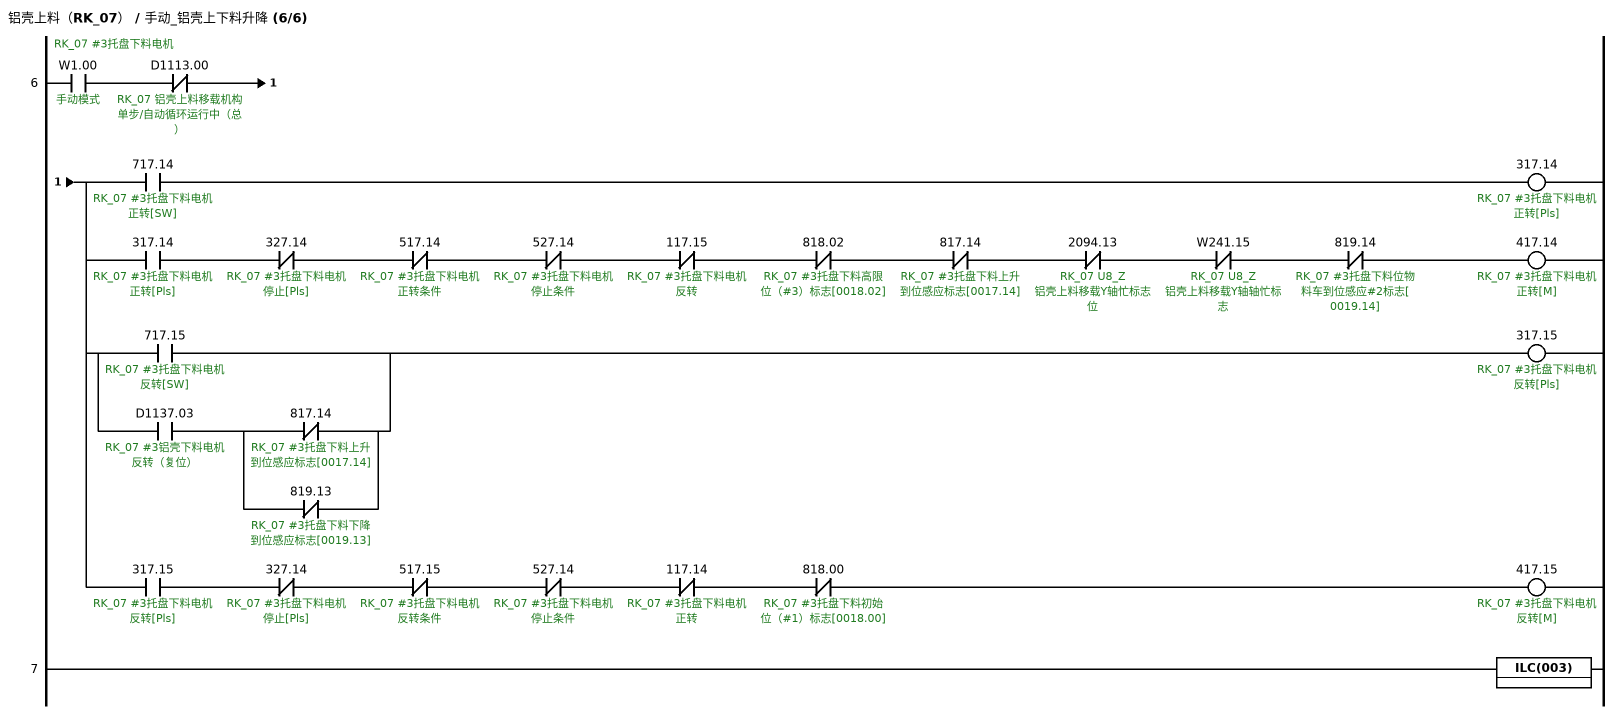
; [picture p576: 铝壳上料（RK_07） / 手动_铝壳上下料升降, rungs 6-7]
; rung 6: RK_07 #3托盘下料电机
LD W1.00  ; 手动模式
ANDNOT D1113.00  ; RK_07 铝壳上料移载机构单步/自动循环运行中（总）
OUT TR0
AND 717.14  ; RK_07 #3托盘下料电机正转[SW]
OUT 317.14  ; RK_07 #3托盘下料电机正转[Pls]
LD TR0
AND 317.14  ; RK_07 #3托盘下料电机正转[Pls]
ANDNOT 327.14  ; RK_07 #3托盘下料电机停止[Pls]
ANDNOT 517.14  ; RK_07 #3托盘下料电机正转条件
ANDNOT 527.14  ; RK_07 #3托盘下料电机停止条件
ANDNOT 117.15  ; RK_07 #3托盘下料电机反转
ANDNOT 818.02  ; RK_07 #3托盘下料高限位（#3）标志[0018.02]
ANDNOT 817.14  ; RK_07 #3托盘下料上升到位感应标志[0017.14]  // 手动模式加此联锁！
ANDNOT 2094.13  ; RK_07 U8_Z 铝壳上料移载Y轴忙标志位
ANDNOT W241.15  ; RK_07 U8_Z 铝壳上料移载Y轴轴忙标志
ANDNOT 819.14  ; RK_07 #3托盘下料位物料车到位感应#2标志[0019.14]
OUT 417.14  ; RK_07 #3托盘下料电机正转[M]
LD TR0
LD 717.15  ; RK_07 #3托盘下料电机反转[SW]
LD D1137.03  ; RK_07 #3铝壳下料电机反转（复位）
LDNOT 817.14  ; RK_07 #3托盘下料上升到位感应标志[0017.14]
ORNOT 819.13  ; RK_07 #3托盘下料下降到位感应标志[0019.13]
ANDLD
ORLD
ANDLD
OUT 317.15  ; RK_07 #3托盘下料电机反转[Pls]
LD TR0
AND 317.15  ; RK_07 #3托盘下料电机反转[Pls]
ANDNOT 327.14  ; RK_07 #3托盘下料电机停止[Pls]
ANDNOT 517.15  ; RK_07 #3托盘下料电机反转条件
ANDNOT 527.14  ; RK_07 #3托盘下料电机停止条件
ANDNOT 117.14  ; RK_07 #3托盘下料电机正转
ANDNOT 818.00  ; RK_07 #3托盘下料初始位（#1）标志[0018.00]
OUT 417.15  ; RK_07 #3托盘下料电机反转[M]
; rung 7
ILC(003)

### Section 自动_铝壳进料

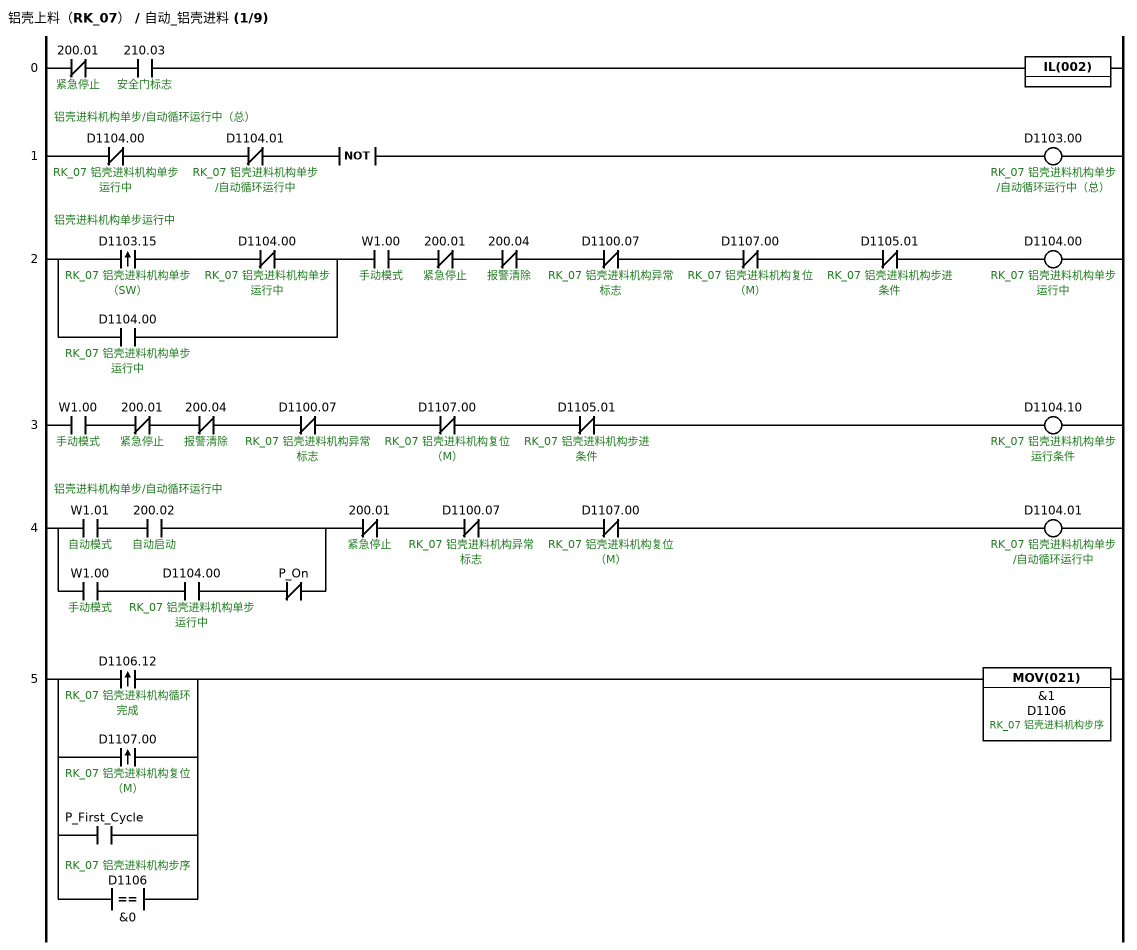
; rung 0
LDNOT 200.01  ; 紧急停止
AND 210.03  ; 安全门标志
IL(002)
; rung 1: 铝壳进料机构单步/自动循环运行中（总）
LDNOT D1104.00  ; RK_07 铝壳进料机构单步运行中
ANDNOT D1104.01  ; RK_07 铝壳进料机构单步/自动循环运行中
NOT(520)
OUT D1103.00  ; RK_07 铝壳进料机构单步/自动循环运行中（总）
; rung 2: 铝壳进料机构单步运行中
@LD D1103.15  ; RK_07 铝壳进料机构单步（SW）
ANDNOT D1104.00  ; RK_07 铝壳进料机构单步运行中
OR D1104.00  ; RK_07 铝壳进料机构单步运行中
AND W1.00  ; 手动模式
ANDNOT 200.01  ; 紧急停止
ANDNOT 200.04  ; 报警清除
ANDNOT D1100.07  ; RK_07 铝壳进料机构异常标志
ANDNOT D1107.00  ; RK_07 铝壳进料机构复位（M）
ANDNOT D1105.01  ; RK_07 铝壳进料机构步进条件
OUT D1104.00  ; RK_07 铝壳进料机构单步运行中
; rung 3
LD W1.00  ; 手动模式
ANDNOT 200.01  ; 紧急停止
ANDNOT 200.04  ; 报警清除
ANDNOT D1100.07  ; RK_07 铝壳进料机构异常标志
ANDNOT D1107.00  ; RK_07 铝壳进料机构复位（M）
ANDNOT D1105.01  ; RK_07 铝壳进料机构步进条件
OUT D1104.10  ; RK_07 铝壳进料机构单步运行条件
; rung 4: 铝壳进料机构单步/自动循环运行中
LD W1.01  ; 自动模式
AND 200.02  ; 自动启动
LD W1.00  ; 手动模式
AND D1104.00  ; RK_07 铝壳进料机构单步运行中
ANDNOT P_On
ORLD
ANDNOT 200.01  ; 紧急停止
ANDNOT D1100.07  ; RK_07 铝壳进料机构异常标志
ANDNOT D1107.00  ; RK_07 铝壳进料机构复位（M）
OUT D1104.01  ; RK_07 铝壳进料机构单步/自动循环运行中
; rung 5
@LD D1106.12  ; RK_07 铝壳进料机构循环完成
@OR D1107.00  ; RK_07 铝壳进料机构复位（M）
OR P_First_Cycle
OR=(300) D1106 &0  ; RK_07 铝壳进料机构步序
MOV(021) &1 D1106  ; RK_07 铝壳进料机构步序

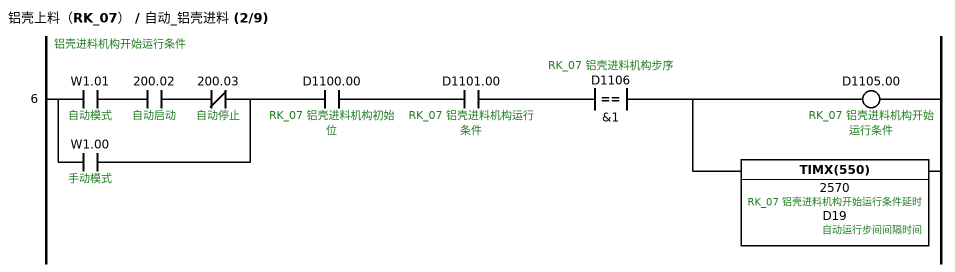
; rung 6: 铝壳进料机构开始运行条件
LD W1.01  ; 自动模式
AND 200.02  ; 自动启动
ANDNOT 200.03  ; 自动停止
OR W1.00  ; 手动模式
AND D1100.00  ; RK_07 铝壳进料机构初始位
AND D1101.00  ; RK_07 铝壳进料机构运行条件
AND=(300) D1106 &1  ; RK_07 铝壳进料机构步序
OUT D1105.00  ; RK_07 铝壳进料机构开始运行条件
TIMX(550) 2570 D19  ; 自动运行步间间隔时间, RK_07 铝壳进料机构开始运行条件延时

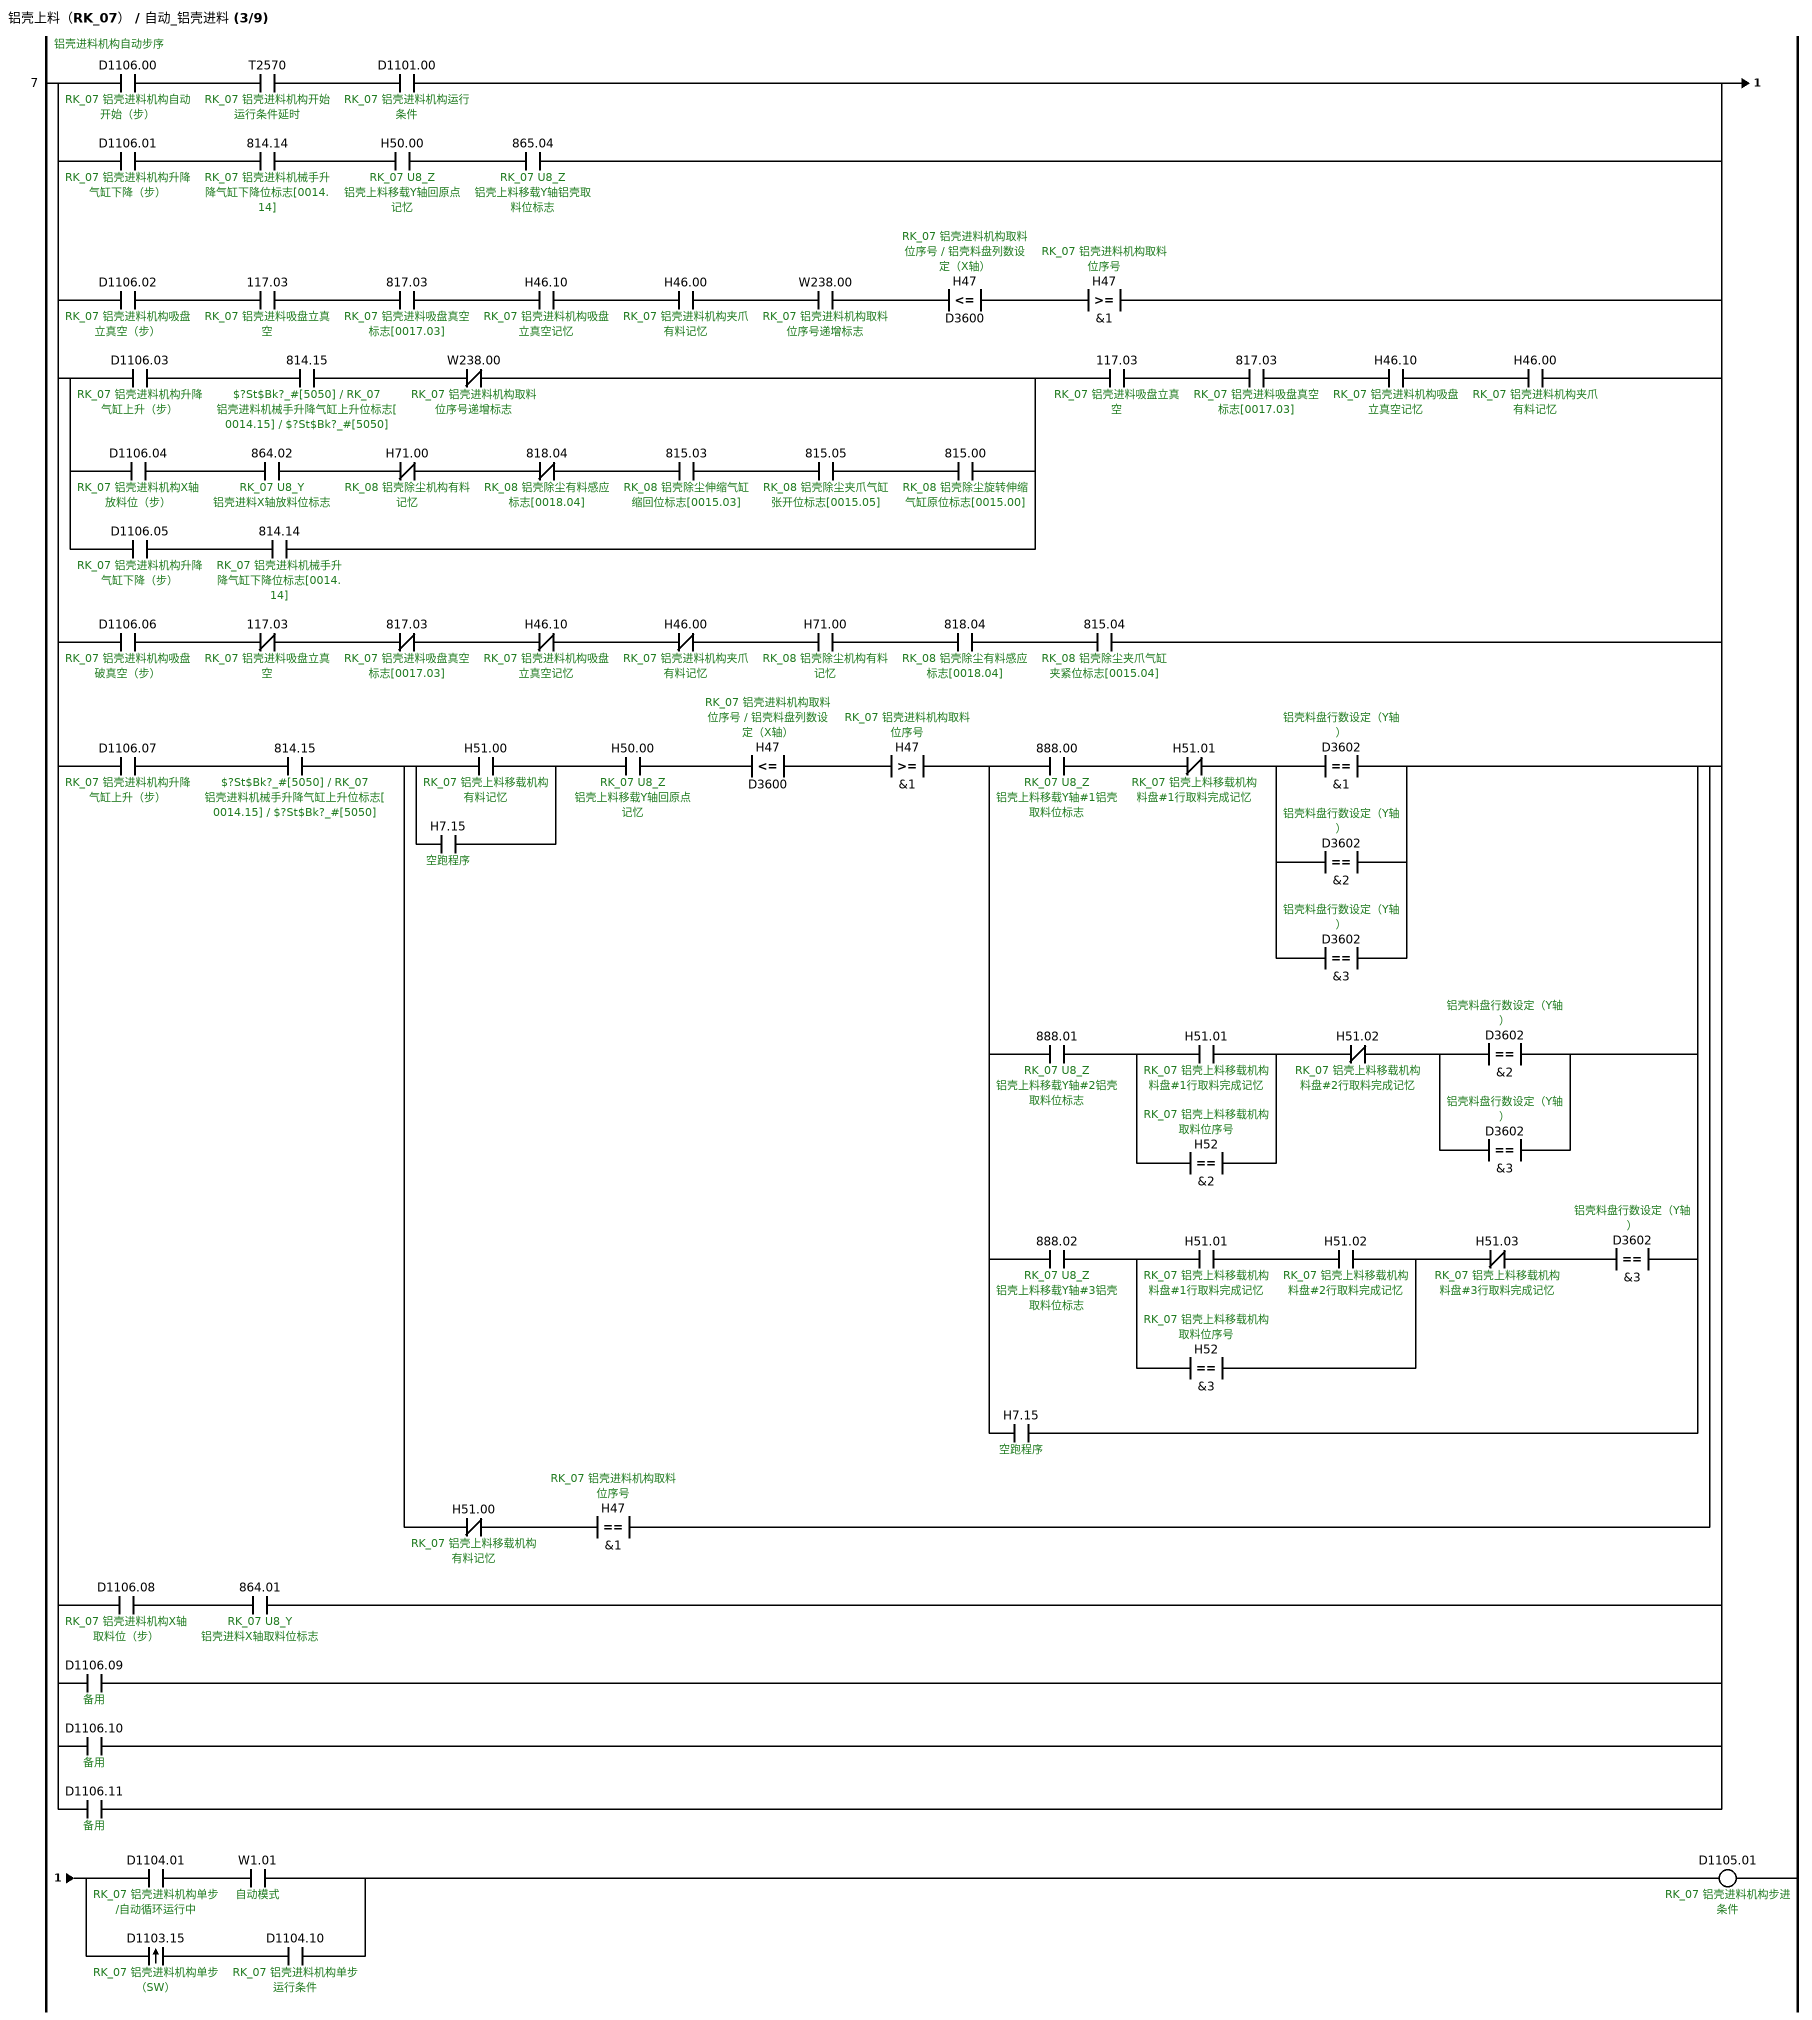
; rung 7: 铝壳进料机构自动步序
LD D1106.00  ; RK_07 铝壳进料机构自动开始（步）
AND T2570  ; RK_07 铝壳进料机构开始运行条件延时
AND D1101.00  ; RK_07 铝壳进料机构运行条件
LD D1106.01  ; RK_07 铝壳进料机构升降气缸下降（步）
AND 814.14  ; RK_07 铝壳进料机械手升降气缸下降位标志[0014.14]
AND H50.00  ; RK_07 U8_Z 铝壳上料移载Y轴回原点记忆
AND 865.04  ; RK_07 U8_Z 铝壳上料移载Y轴铝壳取料位标志
ORLD
LD D1106.02  ; RK_07 铝壳进料机构吸盘立真空（步）
AND 117.03  ; RK_07 铝壳进料吸盘立真空
AND 817.03  ; RK_07 铝壳进料吸盘真空标志[0017.03]
AND H46.10  ; RK_07 铝壳进料机构吸盘立真空记忆
AND H46.00  ; RK_07 铝壳进料机构夹爪有料记忆
AND W238.00  ; RK_07 铝壳进料机构取料位序号递增标志
AND<=(315) H47 D3600  ; RK_07 铝壳进料机构取料位序号, 铝壳料盘列数设定（X轴）
AND>=(325) H47 &1  ; RK_07 铝壳进料机构取料位序号
ORLD
LD D1106.03  ; RK_07 铝壳进料机构升降气缸上升（步）
AND 814.15  ; $?St$Bk?_#[5050] / RK_07 铝壳进料机械手升降气缸上升位标志[0014.15] / $?St$Bk?_#[5050]
ANDNOT W238.00  ; RK_07 铝壳进料机构取料位序号递增标志
LD D1106.04  ; RK_07 铝壳进料机构X轴放料位（步）
AND 864.02  ; RK_07 U8_Y 铝壳进料X轴放料位标志
ANDNOT H71.00  ; RK_08 铝壳除尘机构有料记忆
ANDNOT 818.04  ; RK_08 铝壳除尘有料感应标志[0018.04]
AND 815.03  ; RK_08 铝壳除尘伸缩气缸缩回位标志[0015.03]
AND 815.05  ; RK_08 铝壳除尘夹爪气缸张开位标志[0015.05]
AND 815.00  ; RK_08 铝壳除尘旋转伸缩气缸原位标志[0015.00]
ORLD
LD D1106.05  ; RK_07 铝壳进料机构升降气缸下降（步）
AND 814.14  ; RK_07 铝壳进料机械手升降气缸下降位标志[0014.14]
ORLD
AND 117.03  ; RK_07 铝壳进料吸盘立真空
AND 817.03  ; RK_07 铝壳进料吸盘真空标志[0017.03]
AND H46.10  ; RK_07 铝壳进料机构吸盘立真空记忆
AND H46.00  ; RK_07 铝壳进料机构夹爪有料记忆
ORLD
LD D1106.06  ; RK_07 铝壳进料机构吸盘破真空（步）
ANDNOT 117.03  ; RK_07 铝壳进料吸盘立真空
ANDNOT 817.03  ; RK_07 铝壳进料吸盘真空标志[0017.03]
ANDNOT H46.10  ; RK_07 铝壳进料机构吸盘立真空记忆
ANDNOT H46.00  ; RK_07 铝壳进料机构夹爪有料记忆
AND H71.00  ; RK_08 铝壳除尘机构有料记忆
AND 818.04  ; RK_08 铝壳除尘有料感应标志[0018.04]
AND 815.04  ; RK_08 铝壳除尘夹爪气缸夹紧位标志[0015.04]  // 20181016新增
ORLD
LD D1106.07  ; RK_07 铝壳进料机构升降气缸上升（步）
AND 814.15  ; $?St$Bk?_#[5050] / RK_07 铝壳进料机械手升降气缸上升位标志[0014.15] / $?St$Bk?_#[5050]
LD H51.00  ; RK_07 铝壳上料移载机构有料记忆
OR H7.15  ; 空跑程序
AND H50.00  ; RK_07 U8_Z 铝壳上料移载Y轴回原点记忆
AND<=(315) H47 D3600  ; RK_07 铝壳进料机构取料位序号, 铝壳料盘列数设定（X轴）
AND>=(325) H47 &1  ; RK_07 铝壳进料机构取料位序号
LD 888.00  ; RK_07 U8_Z 铝壳上料移载Y轴#1铝壳取料位标志
ANDNOT H51.01  ; RK_07 铝壳上料移载机构料盘#1行取料完成记忆
LD=(300) D3602 &1  ; 铝壳料盘行数设定（Y轴）
OR=(300) D3602 &2  ; 铝壳料盘行数设定（Y轴）
OR=(300) D3602 &3  ; 铝壳料盘行数设定（Y轴）
ANDLD
LD 888.01  ; RK_07 U8_Z 铝壳上料移载Y轴#2铝壳取料位标志
LD H51.01  ; RK_07 铝壳上料移载机构料盘#1行取料完成记忆
OR=(300) H52 &2  ; RK_07 铝壳上料移载机构取料位序号
ANDLD
ANDNOT H51.02  ; RK_07 铝壳上料移载机构料盘#2行取料完成记忆
LD=(300) D3602 &2  ; 铝壳料盘行数设定（Y轴）
OR=(300) D3602 &3  ; 铝壳料盘行数设定（Y轴）
ANDLD
ORLD
LD 888.02  ; RK_07 U8_Z 铝壳上料移载Y轴#3铝壳取料位标志
LD H51.01  ; RK_07 铝壳上料移载机构料盘#1行取料完成记忆
AND H51.02  ; RK_07 铝壳上料移载机构料盘#2行取料完成记忆
OR=(300) H52 &3  ; RK_07 铝壳上料移载机构取料位序号
ANDLD
ANDNOT H51.03  ; RK_07 铝壳上料移载机构料盘#3行取料完成记忆
AND=(300) D3602 &3  ; 铝壳料盘行数设定（Y轴）
ORLD
OR H7.15  ; 空跑程序
ANDLD
LDNOT H51.00  ; RK_07 铝壳上料移载机构有料记忆
AND=(300) H47 &1  ; RK_07 铝壳进料机构取料位序号
ORLD
ANDLD
ORLD
LD D1106.08  ; RK_07 铝壳进料机构X轴取料位（步）
AND 864.01  ; RK_07 U8_Y 铝壳进料X轴取料位标志
ORLD
OR D1106.09  ; 备用
OR D1106.10  ; 备用
OR D1106.11  ; 备用
LD D1104.01  ; RK_07 铝壳进料机构单步/自动循环运行中
AND W1.01  ; 自动模式
@LD D1103.15  ; RK_07 铝壳进料机构单步（SW）
AND D1104.10  ; RK_07 铝壳进料机构单步运行条件
ORLD
ANDLD
OUT D1105.01  ; RK_07 铝壳进料机构步进条件

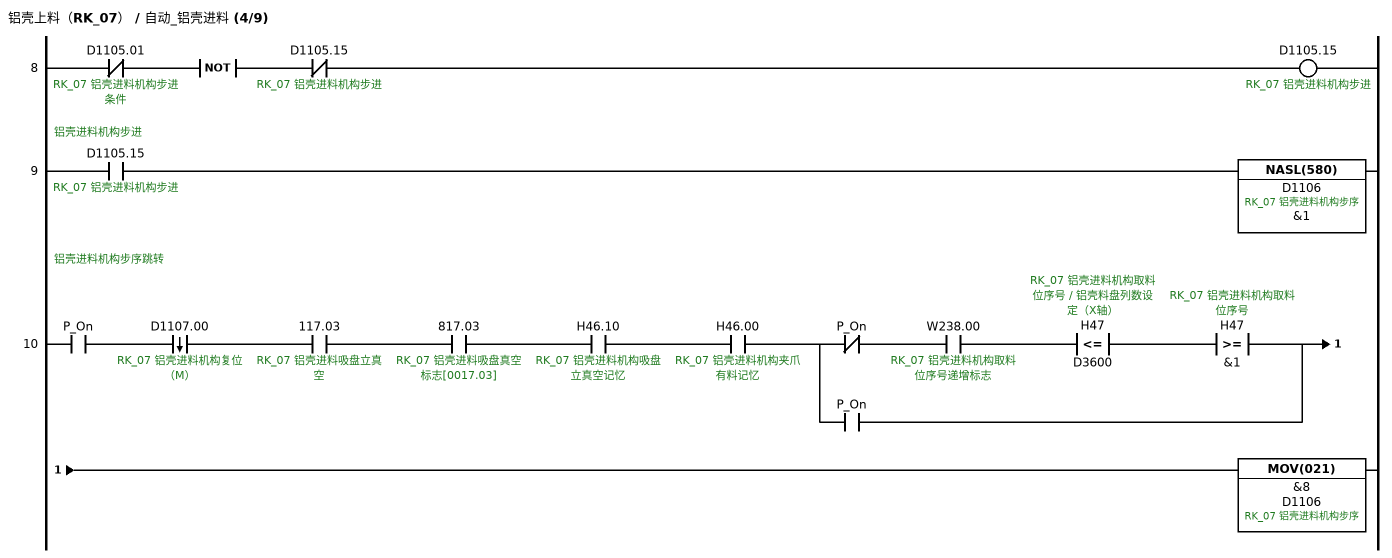
; rung 8
LDNOT D1105.01  ; RK_07 铝壳进料机构步进条件
NOT(520)
ANDNOT D1105.15  ; RK_07 铝壳进料机构步进
OUT D1105.15  ; RK_07 铝壳进料机构步进
; rung 9: 铝壳进料机构步进
LD D1105.15  ; RK_07 铝壳进料机构步进
NASL(580) D1106 &1  ; RK_07 铝壳进料机构步序
; rung 10: 铝壳进料机构步序跳转
LD P_On
%AND D1107.00  ; RK_07 铝壳进料机构复位（M）
AND 117.03  ; RK_07 铝壳进料吸盘立真空
AND 817.03  ; RK_07 铝壳进料吸盘真空标志[0017.03]
AND H46.10  ; RK_07 铝壳进料机构吸盘立真空记忆
AND H46.00  ; RK_07 铝壳进料机构夹爪有料记忆
LDNOT P_On
AND W238.00  ; RK_07 铝壳进料机构取料位序号递增标志
AND<=(315) H47 D3600  ; RK_07 铝壳进料机构取料位序号, 铝壳料盘列数设定（X轴）
AND>=(325) H47 &1  ; RK_07 铝壳进料机构取料位序号
OR P_On
ANDLD
MOV(021) &8 D1106  ; RK_07 铝壳进料机构步序  // RK_07 铝壳进料机构升降气缸上升步（D1106.03）

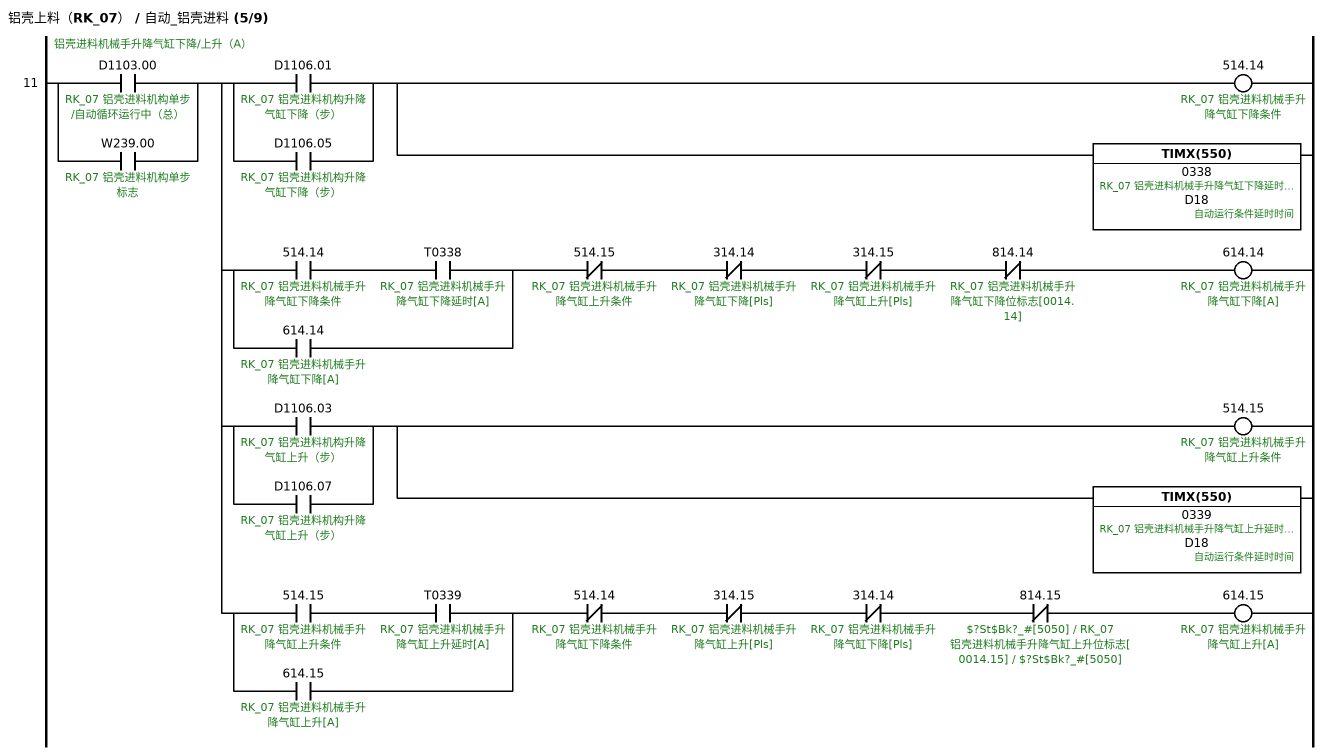
; rung 11: 铝壳进料机械手升降气缸下降/上升（A）
LD D1103.00  ; RK_07 铝壳进料机构单步/自动循环运行中（总）
OR W239.00  ; RK_07 铝壳进料机构单步标志
OUT TR0
LD D1106.01  ; RK_07 铝壳进料机构升降气缸下降（步）
OR D1106.05  ; RK_07 铝壳进料机构升降气缸下降（步）
ANDLD
OUT 514.14  ; RK_07 铝壳进料机械手升降气缸下降条件
TIMX(550) 0338 D18  ; 自动运行条件延时时间, RK_07 铝壳进料机械手升降气缸下降延时[A]
LD TR0
LD 514.14  ; RK_07 铝壳进料机械手升降气缸下降条件
AND T0338  ; RK_07 铝壳进料机械手升降气缸下降延时[A]
OR 614.14  ; RK_07 铝壳进料机械手升降气缸下降[A]
ANDLD
ANDNOT 514.15  ; RK_07 铝壳进料机械手升降气缸上升条件
ANDNOT 314.14  ; RK_07 铝壳进料机械手升降气缸下降[Pls]
ANDNOT 314.15  ; RK_07 铝壳进料机械手升降气缸上升[Pls]
ANDNOT 814.14  ; RK_07 铝壳进料机械手升降气缸下降位标志[0014.14]
OUT 614.14  ; RK_07 铝壳进料机械手升降气缸下降[A]
LD TR0
LD D1106.03  ; RK_07 铝壳进料机构升降气缸上升（步）
OR D1106.07  ; RK_07 铝壳进料机构升降气缸上升（步）
ANDLD
OUT 514.15  ; RK_07 铝壳进料机械手升降气缸上升条件
TIMX(550) 0339 D18  ; 自动运行条件延时时间, RK_07 铝壳进料机械手升降气缸上升延时[A]
LD TR0
LD 514.15  ; RK_07 铝壳进料机械手升降气缸上升条件
AND T0339  ; RK_07 铝壳进料机械手升降气缸上升延时[A]
OR 614.15  ; RK_07 铝壳进料机械手升降气缸上升[A]
ANDLD
ANDNOT 514.14  ; RK_07 铝壳进料机械手升降气缸下降条件
ANDNOT 314.15  ; RK_07 铝壳进料机械手升降气缸上升[Pls]
ANDNOT 314.14  ; RK_07 铝壳进料机械手升降气缸下降[Pls]
ANDNOT 814.15  ; $?St$Bk?_#[5050] / RK_07 铝壳进料机械手升降气缸上升位标志[0014.15] / $?St$Bk?_#[5050]
OUT 614.15  ; RK_07 铝壳进料机械手升降气缸上升[A]

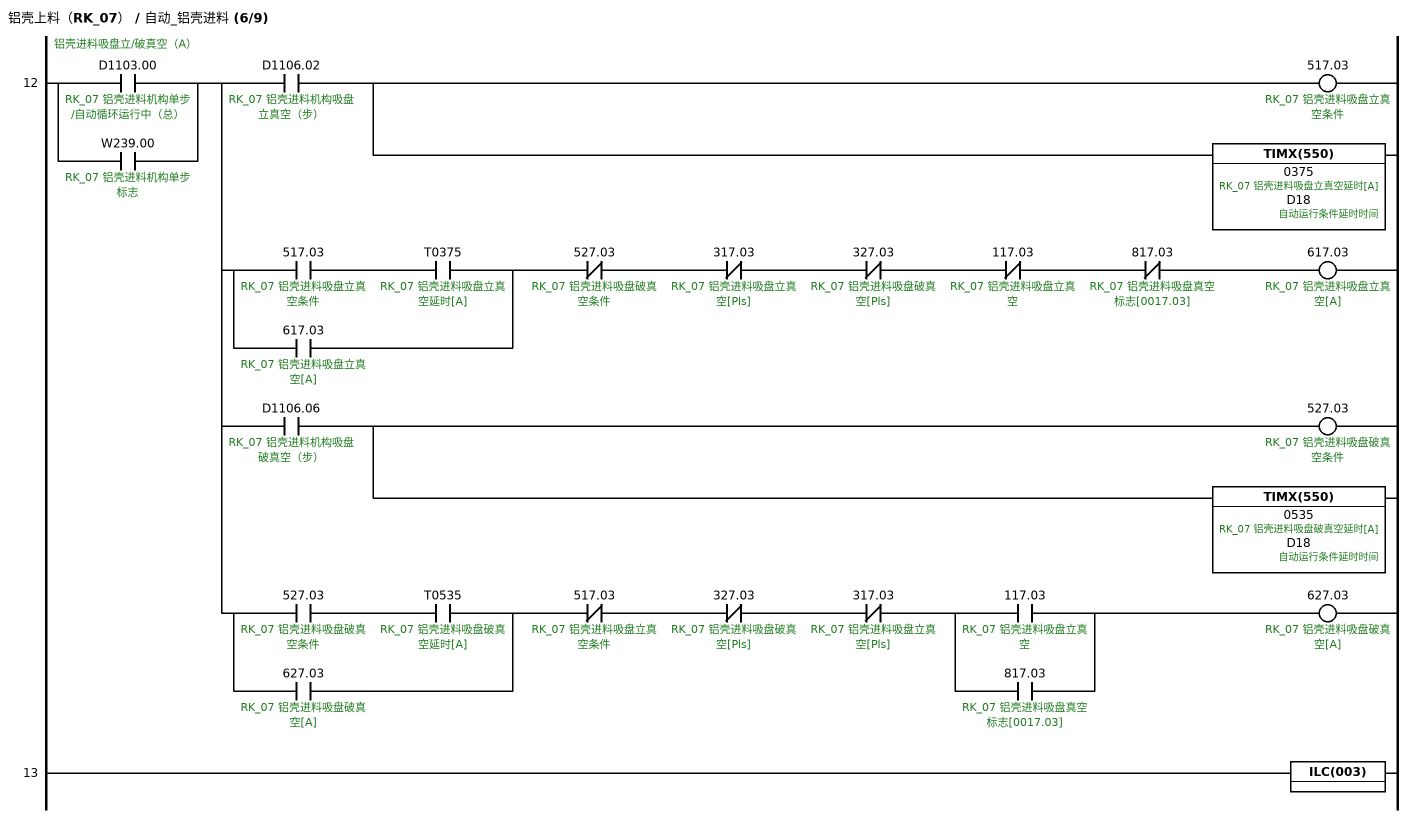
; rung 12: 铝壳进料吸盘立/破真空（A）
LD D1103.00  ; RK_07 铝壳进料机构单步/自动循环运行中（总）
OR W239.00  ; RK_07 铝壳进料机构单步标志
OUT TR0
AND D1106.02  ; RK_07 铝壳进料机构吸盘立真空（步）
OUT 517.03  ; RK_07 铝壳进料吸盘立真空条件
TIMX(550) 0375 D18  ; 自动运行条件延时时间, RK_07 铝壳进料吸盘立真空延时[A]
LD TR0
LD 517.03  ; RK_07 铝壳进料吸盘立真空条件
AND T0375  ; RK_07 铝壳进料吸盘立真空延时[A]
OR 617.03  ; RK_07 铝壳进料吸盘立真空[A]
ANDLD
ANDNOT 527.03  ; RK_07 铝壳进料吸盘破真空条件
ANDNOT 317.03  ; RK_07 铝壳进料吸盘立真空[Pls]
ANDNOT 327.03  ; RK_07 铝壳进料吸盘破真空[Pls]
ANDNOT 117.03  ; RK_07 铝壳进料吸盘立真空
ANDNOT 817.03  ; RK_07 铝壳进料吸盘真空标志[0017.03]
OUT 617.03  ; RK_07 铝壳进料吸盘立真空[A]
LD TR0
AND D1106.06  ; RK_07 铝壳进料机构吸盘破真空（步）
OUT 527.03  ; RK_07 铝壳进料吸盘破真空条件
TIMX(550) 0535 D18  ; 自动运行条件延时时间, RK_07 铝壳进料吸盘破真空延时[A]
LD TR0
LD 527.03  ; RK_07 铝壳进料吸盘破真空条件
AND T0535  ; RK_07 铝壳进料吸盘破真空延时[A]
OR 627.03  ; RK_07 铝壳进料吸盘破真空[A]
ANDLD
ANDNOT 517.03  ; RK_07 铝壳进料吸盘立真空条件
ANDNOT 327.03  ; RK_07 铝壳进料吸盘破真空[Pls]
ANDNOT 317.03  ; RK_07 铝壳进料吸盘立真空[Pls]
LD 117.03  ; RK_07 铝壳进料吸盘立真空
OR 817.03  ; RK_07 铝壳进料吸盘真空标志[0017.03]
ANDLD
OUT 627.03  ; RK_07 铝壳进料吸盘破真空[A]
; rung 13
ILC(003)

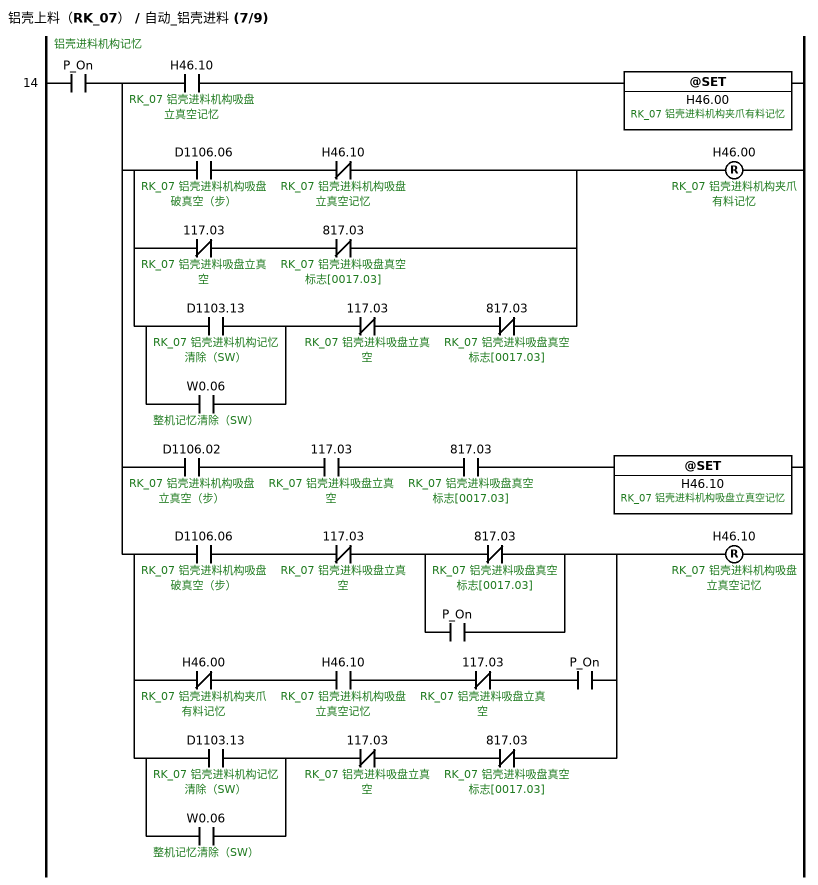
; rung 14: 铝壳进料机构记忆
LD P_On
OUT TR0
AND H46.10  ; RK_07 铝壳进料机构吸盘立真空记忆
@SET H46.00  ; RK_07 铝壳进料机构夹爪有料记忆
LD TR0
LD D1106.06  ; RK_07 铝壳进料机构吸盘破真空（步）
ANDNOT H46.10  ; RK_07 铝壳进料机构吸盘立真空记忆
LDNOT 117.03  ; RK_07 铝壳进料吸盘立真空
ANDNOT 817.03  ; RK_07 铝壳进料吸盘真空标志[0017.03]
ORLD
LD D1103.13  ; RK_07 铝壳进料机构记忆清除（SW）
OR W0.06  ; 整机记忆清除（SW）
ANDNOT 117.03  ; RK_07 铝壳进料吸盘立真空
ANDNOT 817.03  ; RK_07 铝壳进料吸盘真空标志[0017.03]
ORLD
ANDLD
RSET H46.00  ; RK_07 铝壳进料机构夹爪有料记忆
LD TR0
AND D1106.02  ; RK_07 铝壳进料机构吸盘立真空（步）
AND 117.03  ; RK_07 铝壳进料吸盘立真空
AND 817.03  ; RK_07 铝壳进料吸盘真空标志[0017.03]
@SET H46.10  ; RK_07 铝壳进料机构吸盘立真空记忆
LD TR0
LD D1106.06  ; RK_07 铝壳进料机构吸盘破真空（步）
ANDNOT 117.03  ; RK_07 铝壳进料吸盘立真空
LDNOT 817.03  ; RK_07 铝壳进料吸盘真空标志[0017.03]
OR P_On
ANDLD
LDNOT H46.00  ; RK_07 铝壳进料机构夹爪有料记忆
AND H46.10  ; RK_07 铝壳进料机构吸盘立真空记忆
ANDNOT 117.03  ; RK_07 铝壳进料吸盘立真空
AND P_On  // 20181020新增
ORLD
LD D1103.13  ; RK_07 铝壳进料机构记忆清除（SW）
OR W0.06  ; 整机记忆清除（SW）
ANDNOT 117.03  ; RK_07 铝壳进料吸盘立真空
ANDNOT 817.03  ; RK_07 铝壳进料吸盘真空标志[0017.03]
ORLD
ANDLD
RSET H46.10  ; RK_07 铝壳进料机构吸盘立真空记忆

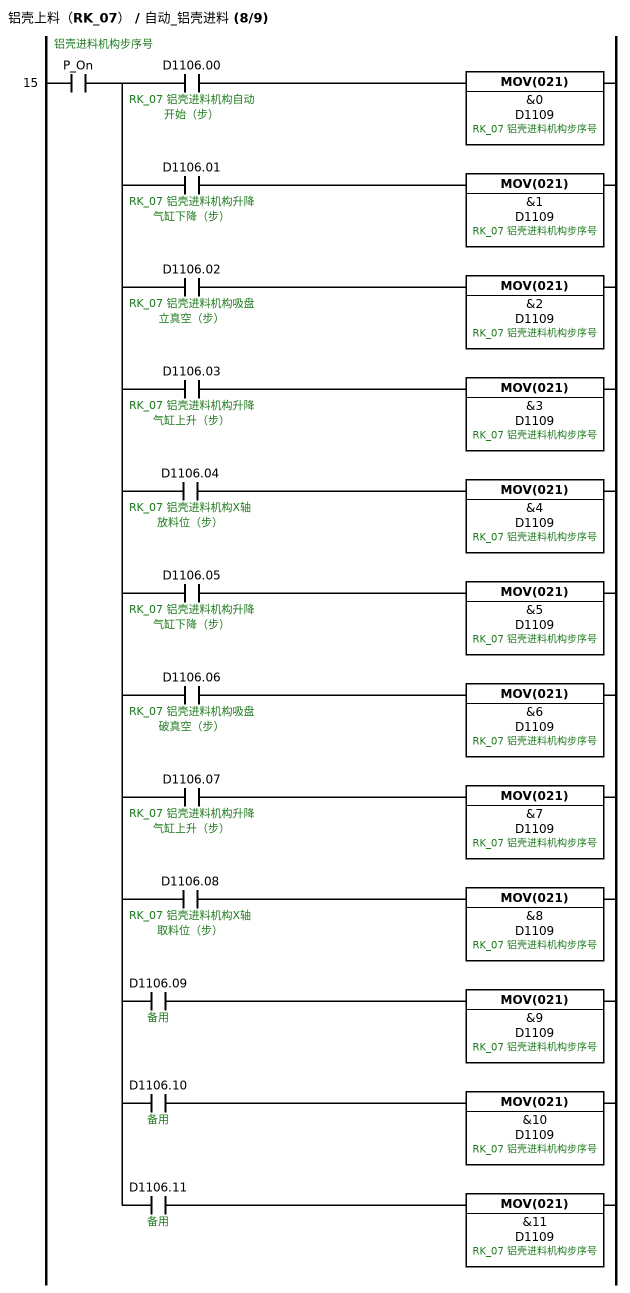
; rung 15: 铝壳进料机构步序号
LD P_On
OUT TR0
AND D1106.00  ; RK_07 铝壳进料机构自动开始（步）
MOV(021) &0 D1109  ; RK_07 铝壳进料机构步序号
LD TR0
AND D1106.01  ; RK_07 铝壳进料机构升降气缸下降（步）
MOV(021) &1 D1109  ; RK_07 铝壳进料机构步序号
LD TR0
AND D1106.02  ; RK_07 铝壳进料机构吸盘立真空（步）
MOV(021) &2 D1109  ; RK_07 铝壳进料机构步序号
LD TR0
AND D1106.03  ; RK_07 铝壳进料机构升降气缸上升（步）
MOV(021) &3 D1109  ; RK_07 铝壳进料机构步序号
LD TR0
AND D1106.04  ; RK_07 铝壳进料机构X轴放料位（步）
MOV(021) &4 D1109  ; RK_07 铝壳进料机构步序号
LD TR0
AND D1106.05  ; RK_07 铝壳进料机构升降气缸下降（步）
MOV(021) &5 D1109  ; RK_07 铝壳进料机构步序号
LD TR0
AND D1106.06  ; RK_07 铝壳进料机构吸盘破真空（步）
MOV(021) &6 D1109  ; RK_07 铝壳进料机构步序号
LD TR0
AND D1106.07  ; RK_07 铝壳进料机构升降气缸上升（步）
MOV(021) &7 D1109  ; RK_07 铝壳进料机构步序号
LD TR0
AND D1106.08  ; RK_07 铝壳进料机构X轴取料位（步）
MOV(021) &8 D1109  ; RK_07 铝壳进料机构步序号
LD TR0
AND D1106.09  ; 备用
MOV(021) &9 D1109  ; RK_07 铝壳进料机构步序号
LD TR0
AND D1106.10  ; 备用
MOV(021) &10 D1109  ; RK_07 铝壳进料机构步序号
LD TR0
AND D1106.11  ; 备用
MOV(021) &11 D1109  ; RK_07 铝壳进料机构步序号

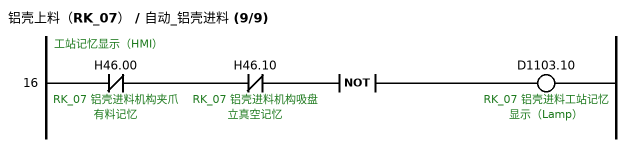
; rung 16: 工站记忆显示（HMI）
LDNOT H46.00  ; RK_07 铝壳进料机构夹爪有料记忆
ANDNOT H46.10  ; RK_07 铝壳进料机构吸盘立真空记忆
NOT(520)
OUT D1103.10  ; RK_07 铝壳进料工站记忆显示（Lamp）

### Section 自动_铝壳上料移载

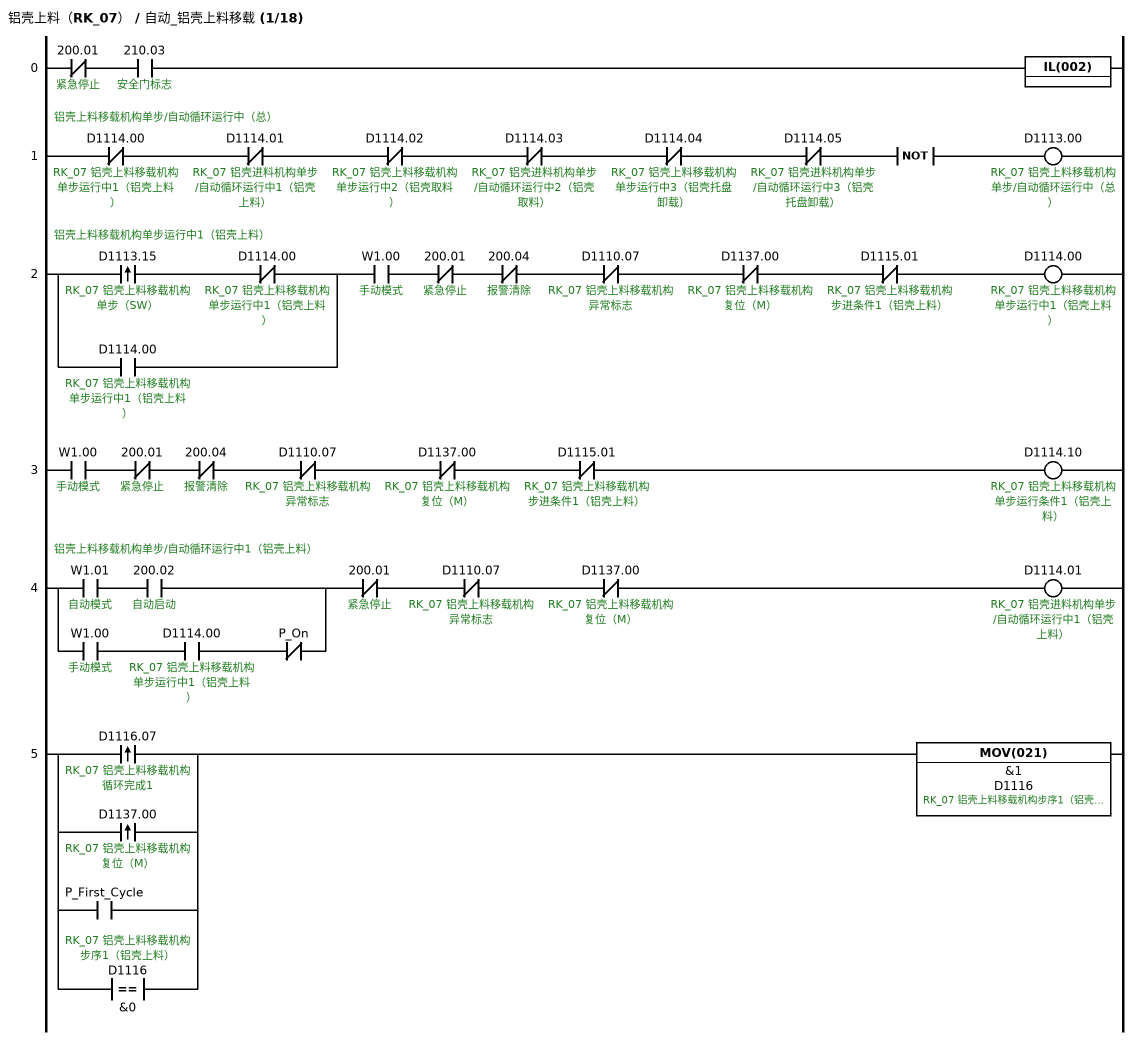
; rung 0
LDNOT 200.01  ; 紧急停止
AND 210.03  ; 安全门标志
IL(002)
; rung 1: 铝壳上料移载机构单步/自动循环运行中（总）
LDNOT D1114.00  ; RK_07 铝壳上料移载机构单步运行中1（铝壳上料）
ANDNOT D1114.01  ; RK_07 铝壳进料机构单步/自动循环运行中1（铝壳上料）
ANDNOT D1114.02  ; RK_07 铝壳上料移载机构单步运行中2（铝壳取料）
ANDNOT D1114.03  ; RK_07 铝壳进料机构单步/自动循环运行中2（铝壳取料）
ANDNOT D1114.04  ; RK_07 铝壳上料移载机构单步运行中3（铝壳托盘卸载）
ANDNOT D1114.05  ; RK_07 铝壳进料机构单步/自动循环运行中3（铝壳托盘卸载）
NOT(520)
OUT D1113.00  ; RK_07 铝壳上料移载机构单步/自动循环运行中（总）
; rung 2: 铝壳上料移载机构单步运行中1（铝壳上料）
@LD D1113.15  ; RK_07 铝壳上料移载机构单步（SW）
ANDNOT D1114.00  ; RK_07 铝壳上料移载机构单步运行中1（铝壳上料）
OR D1114.00  ; RK_07 铝壳上料移载机构单步运行中1（铝壳上料）
AND W1.00  ; 手动模式
ANDNOT 200.01  ; 紧急停止
ANDNOT 200.04  ; 报警清除
ANDNOT D1110.07  ; RK_07 铝壳上料移载机构异常标志
ANDNOT D1137.00  ; RK_07 铝壳上料移载机构复位（M）
ANDNOT D1115.01  ; RK_07 铝壳上料移载机构步进条件1（铝壳上料）
OUT D1114.00  ; RK_07 铝壳上料移载机构单步运行中1（铝壳上料）
; rung 3
LD W1.00  ; 手动模式
ANDNOT 200.01  ; 紧急停止
ANDNOT 200.04  ; 报警清除
ANDNOT D1110.07  ; RK_07 铝壳上料移载机构异常标志
ANDNOT D1137.00  ; RK_07 铝壳上料移载机构复位（M）
ANDNOT D1115.01  ; RK_07 铝壳上料移载机构步进条件1（铝壳上料）
OUT D1114.10  ; RK_07 铝壳上料移载机构单步运行条件1（铝壳上料）
; rung 4: 铝壳上料移载机构单步/自动循环运行中1（铝壳上料）
LD W1.01  ; 自动模式
AND 200.02  ; 自动启动
LD W1.00  ; 手动模式
AND D1114.00  ; RK_07 铝壳上料移载机构单步运行中1（铝壳上料）
ANDNOT P_On
ORLD
ANDNOT 200.01  ; 紧急停止
ANDNOT D1110.07  ; RK_07 铝壳上料移载机构异常标志
ANDNOT D1137.00  ; RK_07 铝壳上料移载机构复位（M）
OUT D1114.01  ; RK_07 铝壳进料机构单步/自动循环运行中1（铝壳上料）
; rung 5
@LD D1116.07  ; RK_07 铝壳上料移载机构循环完成1
@OR D1137.00  ; RK_07 铝壳上料移载机构复位（M）
OR P_First_Cycle
OR=(300) D1116 &0  ; RK_07 铝壳上料移载机构步序1（铝壳上料）
MOV(021) &1 D1116  ; RK_07 铝壳上料移载机构步序1（铝壳上料）

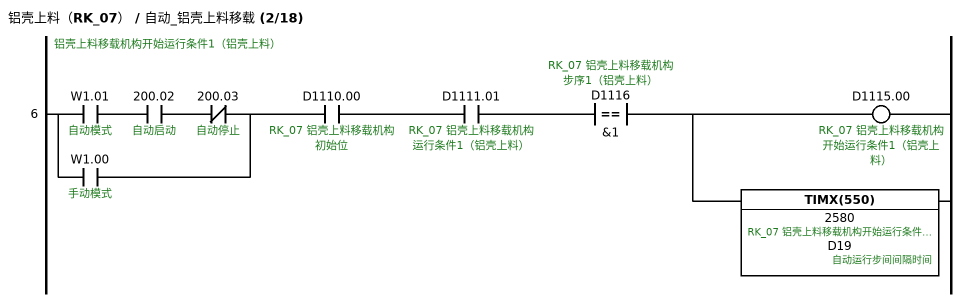
; rung 6: 铝壳上料移载机构开始运行条件1（铝壳上料）
LD W1.01  ; 自动模式
AND 200.02  ; 自动启动
ANDNOT 200.03  ; 自动停止
OR W1.00  ; 手动模式
AND D1110.00  ; RK_07 铝壳上料移载机构初始位
AND D1111.01  ; RK_07 铝壳上料移载机构运行条件1（铝壳上料）
AND=(300) D1116 &1  ; RK_07 铝壳上料移载机构步序1（铝壳上料）
OUT D1115.00  ; RK_07 铝壳上料移载机构开始运行条件1（铝壳上料）
TIMX(550) 2580 D19  ; 自动运行步间间隔时间, RK_07 铝壳上料移载机构开始运行条件1延时（铝壳上料）

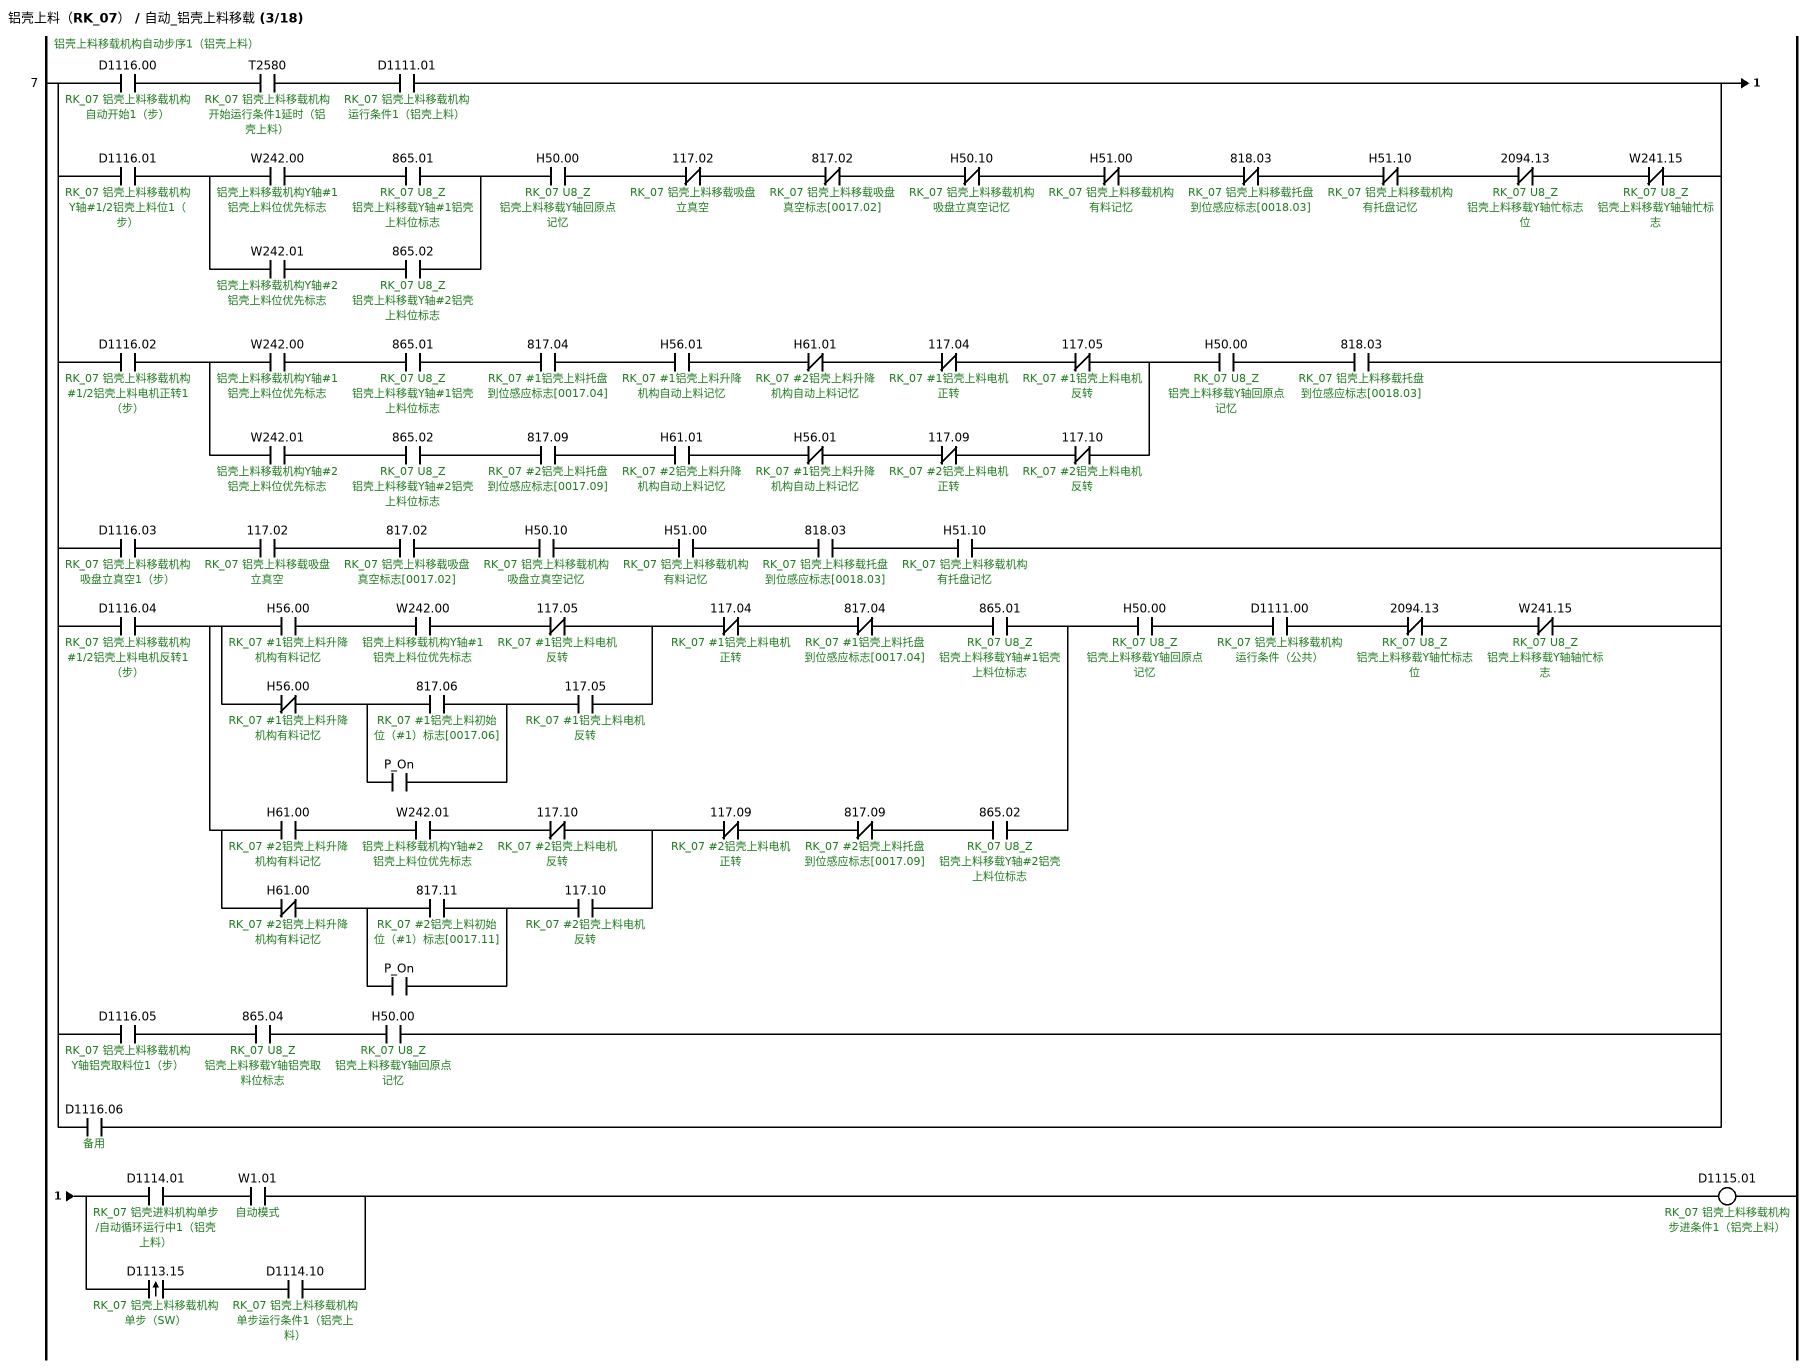
; rung 7: 铝壳上料移载机构自动步序1（铝壳上料）
LD D1116.00  ; RK_07 铝壳上料移载机构自动开始1（步）
AND T2580  ; RK_07 铝壳上料移载机构开始运行条件1延时（铝壳上料）
AND D1111.01  ; RK_07 铝壳上料移载机构运行条件1（铝壳上料）
LD D1116.01  ; RK_07 铝壳上料移载机构Y轴#1/2铝壳上料位1（步）
LD W242.00  ; 铝壳上料移载机构Y轴#1铝壳上料位优先标志
AND 865.01  ; RK_07 U8_Z 铝壳上料移载Y轴#1铝壳上料位标志
LD W242.01  ; 铝壳上料移载机构Y轴#2铝壳上料位优先标志
AND 865.02  ; RK_07 U8_Z 铝壳上料移载Y轴#2铝壳上料位标志
ORLD
ANDLD
AND H50.00  ; RK_07 U8_Z 铝壳上料移载Y轴回原点记忆
ANDNOT 117.02  ; RK_07 铝壳上料移载吸盘立真空
ANDNOT 817.02  ; RK_07 铝壳上料移载吸盘真空标志[0017.02]
ANDNOT H50.10  ; RK_07 铝壳上料移载机构吸盘立真空记忆
ANDNOT H51.00  ; RK_07 铝壳上料移载机构有料记忆
ANDNOT 818.03  ; RK_07 铝壳上料移载托盘到位感应标志[0018.03]
ANDNOT H51.10  ; RK_07 铝壳上料移载机构有托盘记忆
ANDNOT 2094.13  ; RK_07 U8_Z 铝壳上料移载Y轴忙标志位
ANDNOT W241.15  ; RK_07 U8_Z 铝壳上料移载Y轴轴忙标志
ORLD
LD D1116.02  ; RK_07 铝壳上料移载机构#1/2铝壳上料电机正转1（步）
LD W242.00  ; 铝壳上料移载机构Y轴#1铝壳上料位优先标志
AND 865.01  ; RK_07 U8_Z 铝壳上料移载Y轴#1铝壳上料位标志
AND 817.04  ; RK_07 #1铝壳上料托盘到位感应标志[0017.04]
AND H56.01  ; RK_07 #1铝壳上料升降机构自动上料记忆
ANDNOT H61.01  ; RK_07 #2铝壳上料升降机构自动上料记忆
ANDNOT 117.04  ; RK_07 #1铝壳上料电机正转
ANDNOT 117.05  ; RK_07 #1铝壳上料电机反转
LD W242.01  ; 铝壳上料移载机构Y轴#2铝壳上料位优先标志
AND 865.02  ; RK_07 U8_Z 铝壳上料移载Y轴#2铝壳上料位标志
AND 817.09  ; RK_07 #2铝壳上料托盘到位感应标志[0017.09]
AND H61.01  ; RK_07 #2铝壳上料升降机构自动上料记忆
ANDNOT H56.01  ; RK_07 #1铝壳上料升降机构自动上料记忆
ANDNOT 117.09  ; RK_07 #2铝壳上料电机正转
ANDNOT 117.10  ; RK_07 #2铝壳上料电机反转
ORLD
ANDLD
AND H50.00  ; RK_07 U8_Z 铝壳上料移载Y轴回原点记忆
AND 818.03  ; RK_07 铝壳上料移载托盘到位感应标志[0018.03]
ORLD
LD D1116.03  ; RK_07 铝壳上料移载机构吸盘立真空1（步）
AND 117.02  ; RK_07 铝壳上料移载吸盘立真空
AND 817.02  ; RK_07 铝壳上料移载吸盘真空标志[0017.02]
AND H50.10  ; RK_07 铝壳上料移载机构吸盘立真空记忆
AND H51.00  ; RK_07 铝壳上料移载机构有料记忆
AND 818.03  ; RK_07 铝壳上料移载托盘到位感应标志[0018.03]
AND H51.10  ; RK_07 铝壳上料移载机构有托盘记忆
ORLD
LD D1116.04  ; RK_07 铝壳上料移载机构#1/2铝壳上料电机反转1（步）
LD H56.00  ; RK_07 #1铝壳上料升降机构有料记忆
AND W242.00  ; 铝壳上料移载机构Y轴#1铝壳上料位优先标志
ANDNOT 117.05  ; RK_07 #1铝壳上料电机反转
LDNOT H56.00  ; RK_07 #1铝壳上料升降机构有料记忆  // RK_07 #1铝壳上料升降机构最后一个托盘被上料移载抓取之后，#1铝壳上料升降电机反转到#1铝壳上料初始位（#1）感应信号停止！
LD 817.06  ; RK_07 #1铝壳上料初始位（#1）标志[0017.06]
OR P_On
ANDLD
AND 117.05  ; RK_07 #1铝壳上料电机反转
ORLD
ANDNOT 117.04  ; RK_07 #1铝壳上料电机正转
ANDNOT 817.04  ; RK_07 #1铝壳上料托盘到位感应标志[0017.04]
AND 865.01  ; RK_07 U8_Z 铝壳上料移载Y轴#1铝壳上料位标志
LD H61.00  ; RK_07 #2铝壳上料升降机构有料记忆
AND W242.01  ; 铝壳上料移载机构Y轴#2铝壳上料位优先标志
ANDNOT 117.10  ; RK_07 #2铝壳上料电机反转
LDNOT H61.00  ; RK_07 #2铝壳上料升降机构有料记忆  // RK_07 #2铝壳上料升降机构最后一个托盘被上料移载抓取之后，#2铝壳上料升降电机反转到#2铝壳上料初始位（#1）感应信号停止！
LD 817.11  ; RK_07 #2铝壳上料初始位（#1）标志[0017.11]
OR P_On
ANDLD
AND 117.10  ; RK_07 #2铝壳上料电机反转
ORLD
ANDNOT 117.09  ; RK_07 #2铝壳上料电机正转
ANDNOT 817.09  ; RK_07 #2铝壳上料托盘到位感应标志[0017.09]
AND 865.02  ; RK_07 U8_Z 铝壳上料移载Y轴#2铝壳上料位标志
ORLD
ANDLD
AND H50.00  ; RK_07 U8_Z 铝壳上料移载Y轴回原点记忆
AND D1111.00  ; RK_07 铝壳上料移载机构运行条件（公共）
ANDNOT 2094.13  ; RK_07 U8_Z 铝壳上料移载Y轴忙标志位
ANDNOT W241.15  ; RK_07 U8_Z 铝壳上料移载Y轴轴忙标志
ORLD
LD D1116.05  ; RK_07 铝壳上料移载机构Y轴铝壳取料位1（步）
AND 865.04  ; RK_07 U8_Z 铝壳上料移载Y轴铝壳取料位标志
AND H50.00  ; RK_07 U8_Z 铝壳上料移载Y轴回原点记忆
ORLD
OR D1116.06  ; 备用
LD D1114.01  ; RK_07 铝壳进料机构单步/自动循环运行中1（铝壳上料）
AND W1.01  ; 自动模式
@LD D1113.15  ; RK_07 铝壳上料移载机构单步（SW）
AND D1114.10  ; RK_07 铝壳上料移载机构单步运行条件1（铝壳上料）
ORLD
ANDLD
OUT D1115.01  ; RK_07 铝壳上料移载机构步进条件1（铝壳上料）

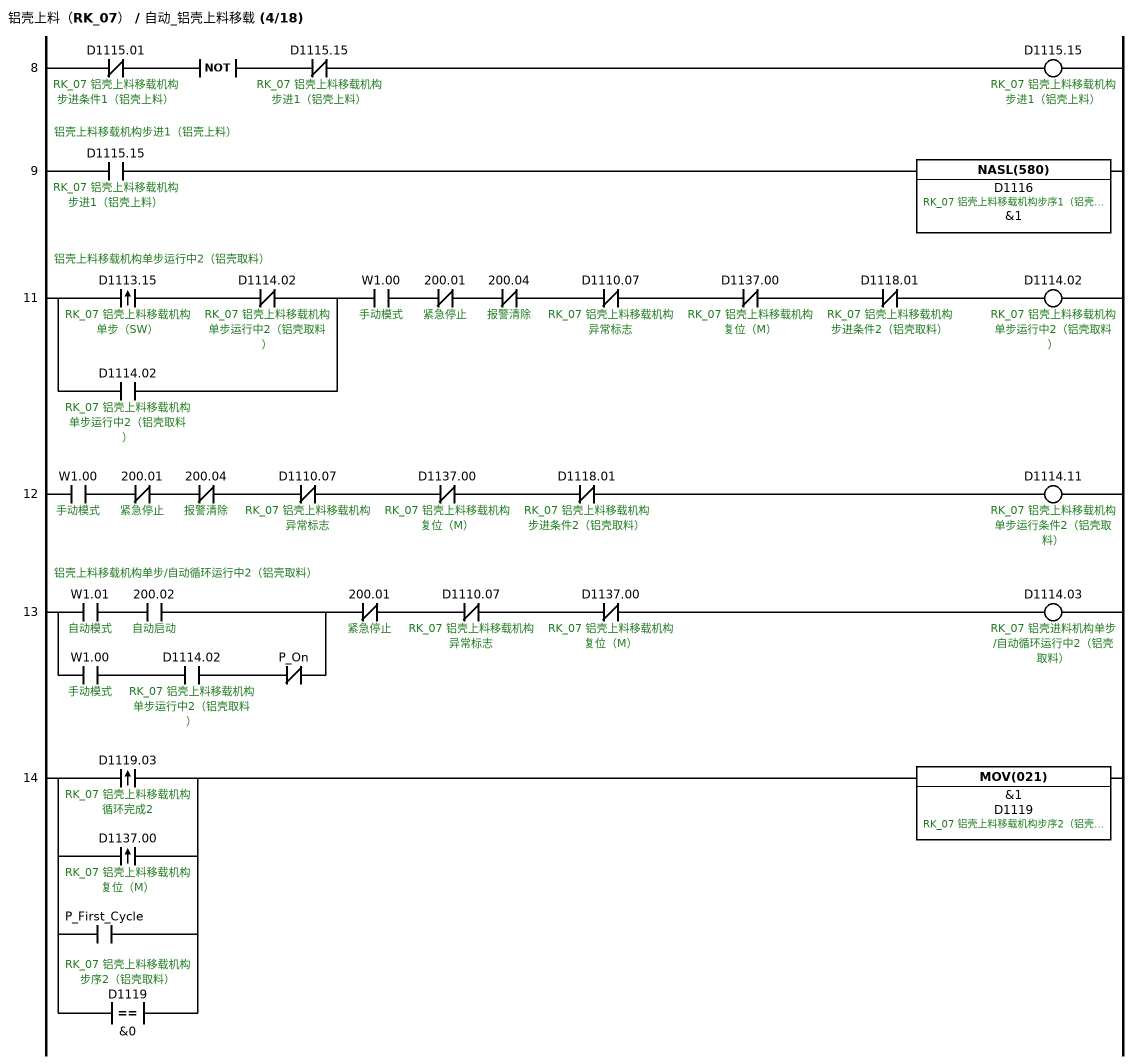
; rung 8
LDNOT D1115.01  ; RK_07 铝壳上料移载机构步进条件1（铝壳上料）
NOT(520)
ANDNOT D1115.15  ; RK_07 铝壳上料移载机构步进1（铝壳上料）
OUT D1115.15  ; RK_07 铝壳上料移载机构步进1（铝壳上料）
; rung 9: 铝壳上料移载机构步进1（铝壳上料）
LD D1115.15  ; RK_07 铝壳上料移载机构步进1（铝壳上料）
NASL(580) D1116 &1  ; RK_07 铝壳上料移载机构步序1（铝壳上料）
; rung 10: 铝壳上料移载机构步序跳转1（铝壳上料）
; rung 11: 铝壳上料移载机构单步运行中2（铝壳取料）
@LD D1113.15  ; RK_07 铝壳上料移载机构单步（SW）
ANDNOT D1114.02  ; RK_07 铝壳上料移载机构单步运行中2（铝壳取料）
OR D1114.02  ; RK_07 铝壳上料移载机构单步运行中2（铝壳取料）
AND W1.00  ; 手动模式
ANDNOT 200.01  ; 紧急停止
ANDNOT 200.04  ; 报警清除
ANDNOT D1110.07  ; RK_07 铝壳上料移载机构异常标志
ANDNOT D1137.00  ; RK_07 铝壳上料移载机构复位（M）
ANDNOT D1118.01  ; RK_07 铝壳上料移载机构步进条件2（铝壳取料）
OUT D1114.02  ; RK_07 铝壳上料移载机构单步运行中2（铝壳取料）
; rung 12
LD W1.00  ; 手动模式
ANDNOT 200.01  ; 紧急停止
ANDNOT 200.04  ; 报警清除
ANDNOT D1110.07  ; RK_07 铝壳上料移载机构异常标志
ANDNOT D1137.00  ; RK_07 铝壳上料移载机构复位（M）
ANDNOT D1118.01  ; RK_07 铝壳上料移载机构步进条件2（铝壳取料）
OUT D1114.11  ; RK_07 铝壳上料移载机构单步运行条件2（铝壳取料）
; rung 13: 铝壳上料移载机构单步/自动循环运行中2（铝壳取料）
LD W1.01  ; 自动模式
AND 200.02  ; 自动启动
LD W1.00  ; 手动模式
AND D1114.02  ; RK_07 铝壳上料移载机构单步运行中2（铝壳取料）
ANDNOT P_On
ORLD
ANDNOT 200.01  ; 紧急停止
ANDNOT D1110.07  ; RK_07 铝壳上料移载机构异常标志
ANDNOT D1137.00  ; RK_07 铝壳上料移载机构复位（M）
OUT D1114.03  ; RK_07 铝壳进料机构单步/自动循环运行中2（铝壳取料）
; rung 14
@LD D1119.03  ; RK_07 铝壳上料移载机构循环完成2
@OR D1137.00  ; RK_07 铝壳上料移载机构复位（M）
OR P_First_Cycle
OR=(300) D1119 &0  ; RK_07 铝壳上料移载机构步序2（铝壳取料）
MOV(021) &1 D1119  ; RK_07 铝壳上料移载机构步序2（铝壳取料）

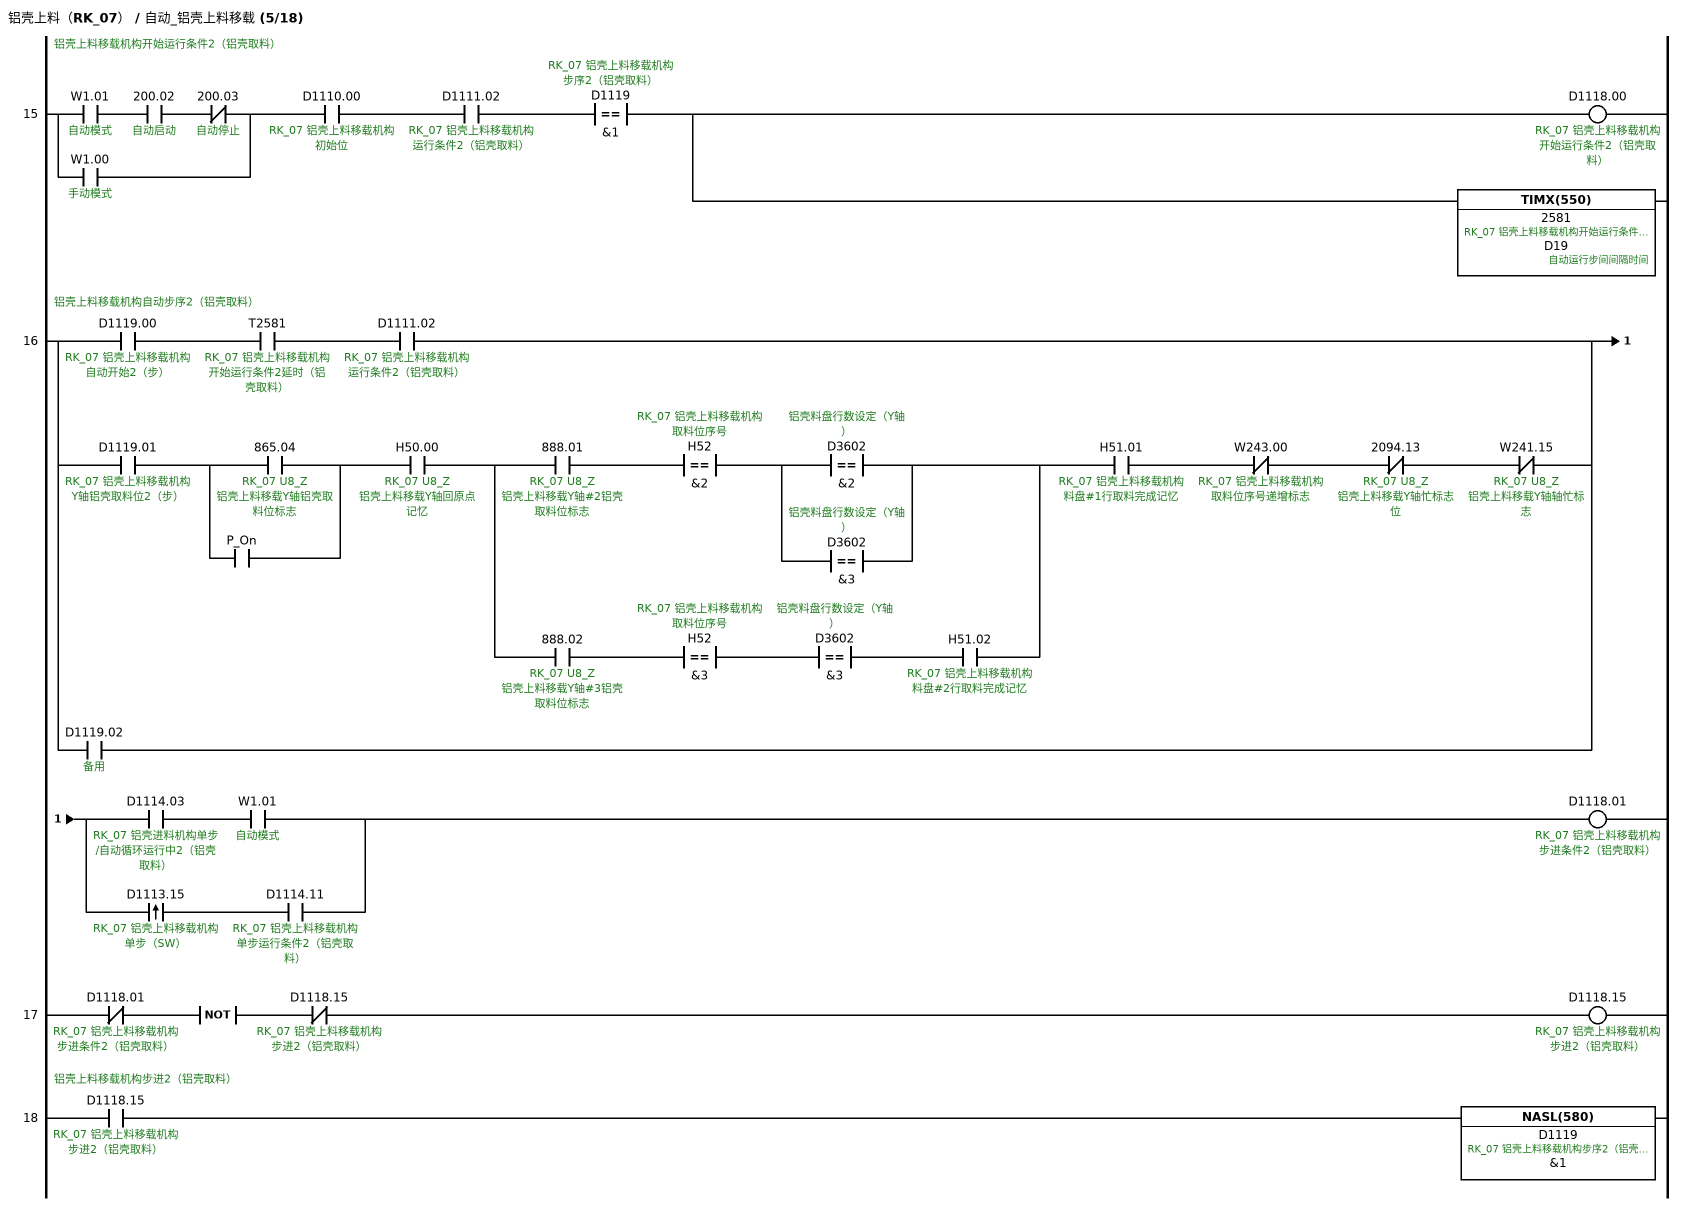
; rung 15: 铝壳上料移载机构开始运行条件2（铝壳取料）
LD W1.01  ; 自动模式
AND 200.02  ; 自动启动
ANDNOT 200.03  ; 自动停止
OR W1.00  ; 手动模式
AND D1110.00  ; RK_07 铝壳上料移载机构初始位
AND D1111.02  ; RK_07 铝壳上料移载机构运行条件2（铝壳取料）
AND=(300) D1119 &1  ; RK_07 铝壳上料移载机构步序2（铝壳取料）
OUT D1118.00  ; RK_07 铝壳上料移载机构开始运行条件2（铝壳取料）
TIMX(550) 2581 D19  ; 自动运行步间间隔时间, RK_07 铝壳上料移载机构开始运行条件2延时（铝壳取料）
; rung 16: 铝壳上料移载机构自动步序2（铝壳取料）
LD D1119.00  ; RK_07 铝壳上料移载机构自动开始2（步）
AND T2581  ; RK_07 铝壳上料移载机构开始运行条件2延时（铝壳取料）
AND D1111.02  ; RK_07 铝壳上料移载机构运行条件2（铝壳取料）
LD D1119.01  ; RK_07 铝壳上料移载机构Y轴铝壳取料位2（步）
LD 865.04  ; RK_07 U8_Z 铝壳上料移载Y轴铝壳取料位标志
OR P_On
ANDLD
AND H50.00  ; RK_07 U8_Z 铝壳上料移载Y轴回原点记忆
LD 888.01  ; RK_07 U8_Z 铝壳上料移载Y轴#2铝壳取料位标志
AND=(300) H52 &2  ; RK_07 铝壳上料移载机构取料位序号
LD=(300) D3602 &2  ; 铝壳料盘行数设定（Y轴）
OR=(300) D3602 &3  ; 铝壳料盘行数设定（Y轴）
ANDLD
LD 888.02  ; RK_07 U8_Z 铝壳上料移载Y轴#3铝壳取料位标志
AND=(300) H52 &3  ; RK_07 铝壳上料移载机构取料位序号
AND=(300) D3602 &3  ; 铝壳料盘行数设定（Y轴）
AND H51.02  ; RK_07 铝壳上料移载机构料盘#2行取料完成记忆
ORLD
ANDLD
AND H51.01  ; RK_07 铝壳上料移载机构料盘#1行取料完成记忆
ANDNOT W243.00  ; RK_07 铝壳上料移载机构取料位序号递增标志
ANDNOT 2094.13  ; RK_07 U8_Z 铝壳上料移载Y轴忙标志位
ANDNOT W241.15  ; RK_07 U8_Z 铝壳上料移载Y轴轴忙标志
ORLD
OR D1119.02  ; 备用
LD D1114.03  ; RK_07 铝壳进料机构单步/自动循环运行中2（铝壳取料）
AND W1.01  ; 自动模式
@LD D1113.15  ; RK_07 铝壳上料移载机构单步（SW）
AND D1114.11  ; RK_07 铝壳上料移载机构单步运行条件2（铝壳取料）
ORLD
ANDLD
OUT D1118.01  ; RK_07 铝壳上料移载机构步进条件2（铝壳取料）
; rung 17
LDNOT D1118.01  ; RK_07 铝壳上料移载机构步进条件2（铝壳取料）
NOT(520)
ANDNOT D1118.15  ; RK_07 铝壳上料移载机构步进2（铝壳取料）
OUT D1118.15  ; RK_07 铝壳上料移载机构步进2（铝壳取料）
; rung 18: 铝壳上料移载机构步进2（铝壳取料）
LD D1118.15  ; RK_07 铝壳上料移载机构步进2（铝壳取料）
NASL(580) D1119 &1  ; RK_07 铝壳上料移载机构步序2（铝壳取料）
; rung 19: 铝壳上料移载机构步序跳转2（铝壳取料）

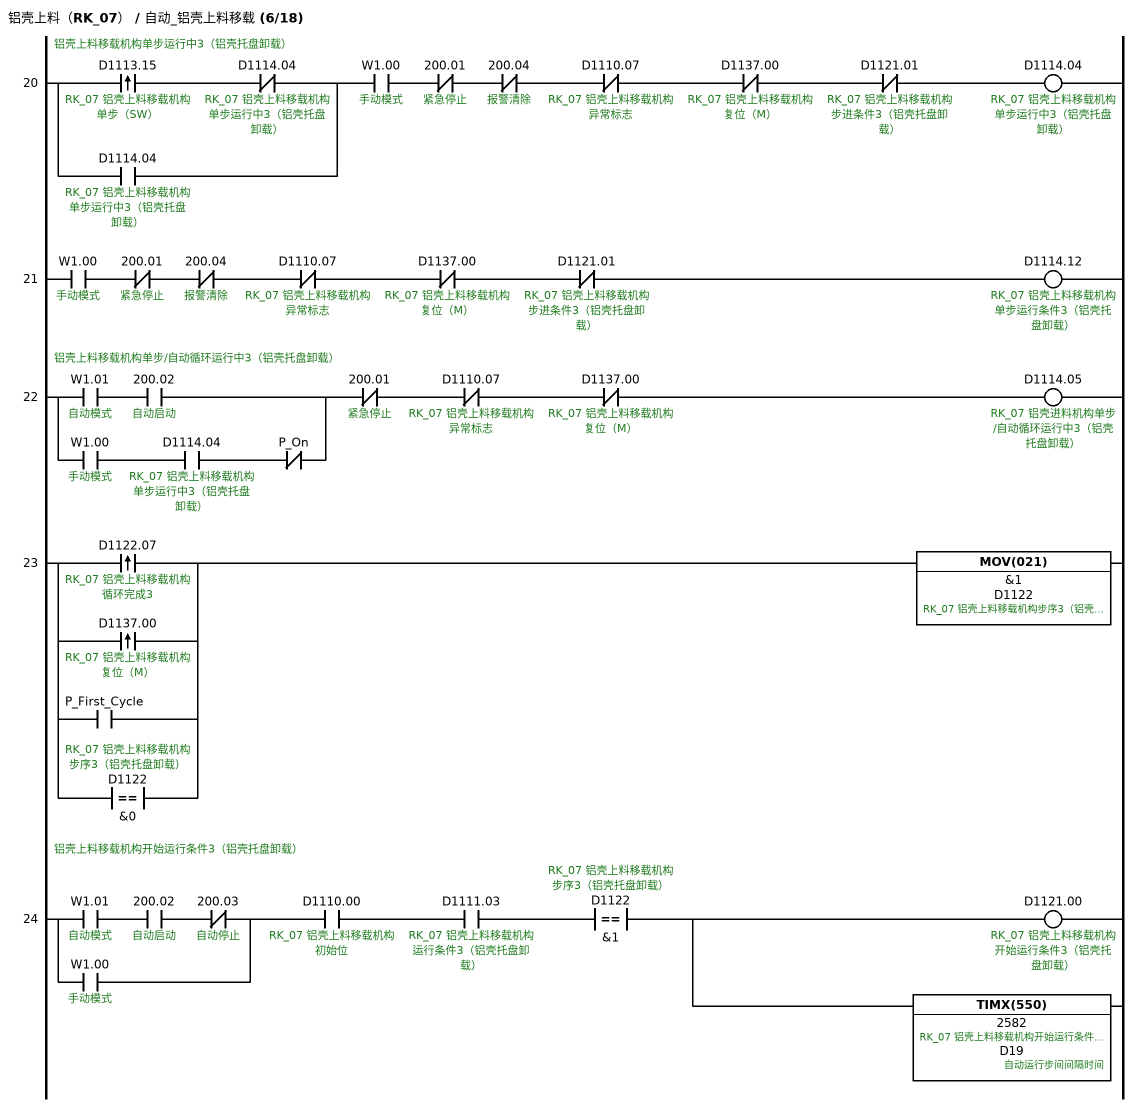
; rung 20: 铝壳上料移载机构单步运行中3（铝壳托盘卸载）
@LD D1113.15  ; RK_07 铝壳上料移载机构单步（SW）
ANDNOT D1114.04  ; RK_07 铝壳上料移载机构单步运行中3（铝壳托盘卸载）
OR D1114.04  ; RK_07 铝壳上料移载机构单步运行中3（铝壳托盘卸载）
AND W1.00  ; 手动模式
ANDNOT 200.01  ; 紧急停止
ANDNOT 200.04  ; 报警清除
ANDNOT D1110.07  ; RK_07 铝壳上料移载机构异常标志
ANDNOT D1137.00  ; RK_07 铝壳上料移载机构复位（M）
ANDNOT D1121.01  ; RK_07 铝壳上料移载机构步进条件3（铝壳托盘卸载）
OUT D1114.04  ; RK_07 铝壳上料移载机构单步运行中3（铝壳托盘卸载）
; rung 21
LD W1.00  ; 手动模式
ANDNOT 200.01  ; 紧急停止
ANDNOT 200.04  ; 报警清除
ANDNOT D1110.07  ; RK_07 铝壳上料移载机构异常标志
ANDNOT D1137.00  ; RK_07 铝壳上料移载机构复位（M）
ANDNOT D1121.01  ; RK_07 铝壳上料移载机构步进条件3（铝壳托盘卸载）
OUT D1114.12  ; RK_07 铝壳上料移载机构单步运行条件3（铝壳托盘卸载）
; rung 22: 铝壳上料移载机构单步/自动循环运行中3（铝壳托盘卸载）
LD W1.01  ; 自动模式
AND 200.02  ; 自动启动
LD W1.00  ; 手动模式
AND D1114.04  ; RK_07 铝壳上料移载机构单步运行中3（铝壳托盘卸载）
ANDNOT P_On
ORLD
ANDNOT 200.01  ; 紧急停止
ANDNOT D1110.07  ; RK_07 铝壳上料移载机构异常标志
ANDNOT D1137.00  ; RK_07 铝壳上料移载机构复位（M）
OUT D1114.05  ; RK_07 铝壳进料机构单步/自动循环运行中3（铝壳托盘卸载）
; rung 23
@LD D1122.07  ; RK_07 铝壳上料移载机构循环完成3
@OR D1137.00  ; RK_07 铝壳上料移载机构复位（M）
OR P_First_Cycle
OR=(300) D1122 &0  ; RK_07 铝壳上料移载机构步序3（铝壳托盘卸载）
MOV(021) &1 D1122  ; RK_07 铝壳上料移载机构步序3（铝壳托盘卸载）
; rung 24: 铝壳上料移载机构开始运行条件3（铝壳托盘卸载）
LD W1.01  ; 自动模式
AND 200.02  ; 自动启动
ANDNOT 200.03  ; 自动停止
OR W1.00  ; 手动模式
AND D1110.00  ; RK_07 铝壳上料移载机构初始位
AND D1111.03  ; RK_07 铝壳上料移载机构运行条件3（铝壳托盘卸载）
AND=(300) D1122 &1  ; RK_07 铝壳上料移载机构步序3（铝壳托盘卸载）
OUT D1121.00  ; RK_07 铝壳上料移载机构开始运行条件3（铝壳托盘卸载）
TIMX(550) 2582 D19  ; 自动运行步间间隔时间, RK_07 铝壳上料移载机构开始运行条件3延时（铝壳托盘卸载）

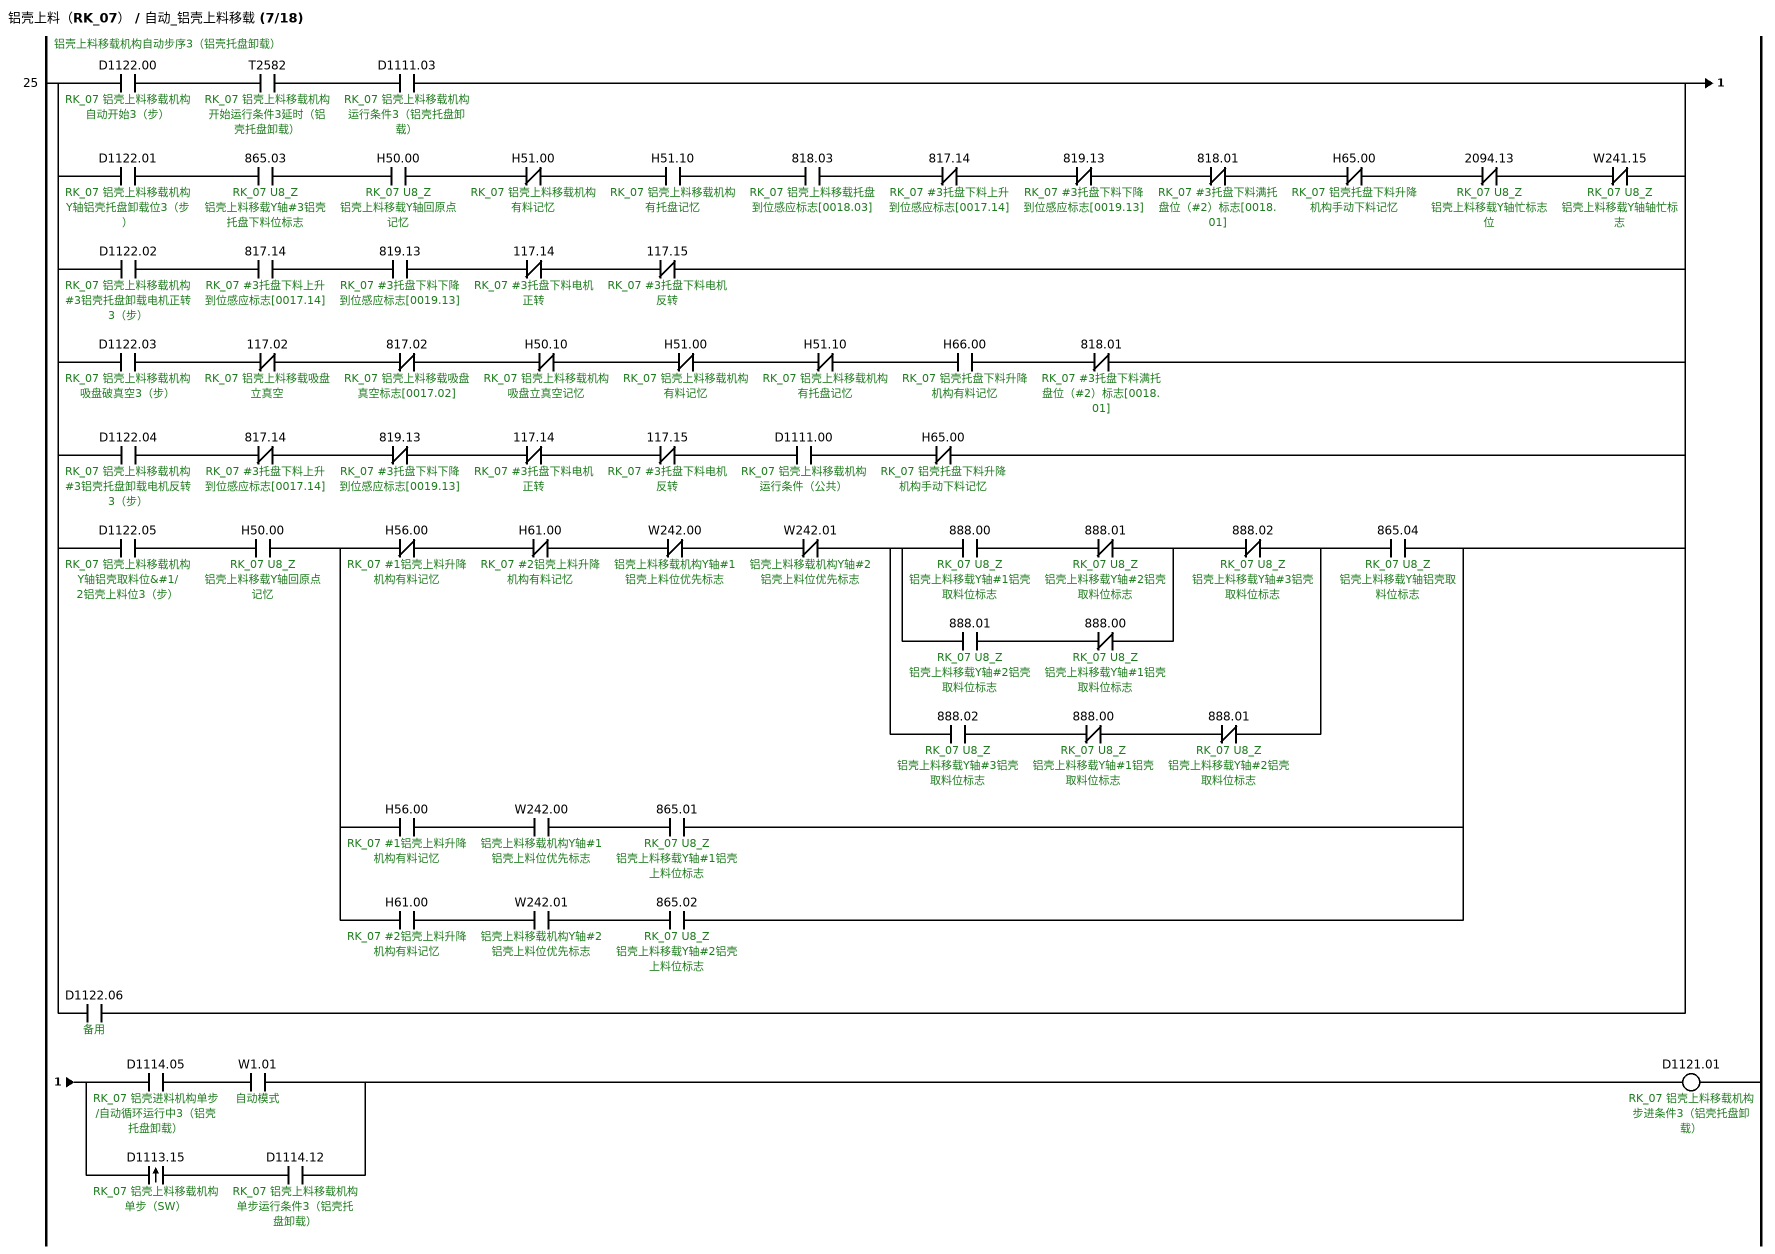
; rung 25: 铝壳上料移载机构自动步序3（铝壳托盘卸载）
LD D1122.00  ; RK_07 铝壳上料移载机构自动开始3（步）
AND T2582  ; RK_07 铝壳上料移载机构开始运行条件3延时（铝壳托盘卸载）
AND D1111.03  ; RK_07 铝壳上料移载机构运行条件3（铝壳托盘卸载）
LD D1122.01  ; RK_07 铝壳上料移载机构Y轴铝壳托盘卸载位3（步）
AND 865.03  ; RK_07 U8_Z 铝壳上料移载Y轴#3铝壳托盘下料位标志
AND H50.00  ; RK_07 U8_Z 铝壳上料移载Y轴回原点记忆
ANDNOT H51.00  ; RK_07 铝壳上料移载机构有料记忆
AND H51.10  ; RK_07 铝壳上料移载机构有托盘记忆
AND 818.03  ; RK_07 铝壳上料移载托盘到位感应标志[0018.03]
ANDNOT 817.14  ; RK_07 #3托盘下料上升到位感应标志[0017.14]
ANDNOT 819.13  ; RK_07 #3托盘下料下降到位感应标志[0019.13]
ANDNOT 818.01  ; RK_07 #3托盘下料满托盘位（#2）标志[0018.01]
ANDNOT H65.00  ; RK_07 铝壳托盘下料升降机构手动下料记忆
ANDNOT 2094.13  ; RK_07 U8_Z 铝壳上料移载Y轴忙标志位
ANDNOT W241.15  ; RK_07 U8_Z 铝壳上料移载Y轴轴忙标志
ORLD
LD D1122.02  ; RK_07 铝壳上料移载机构#3铝壳托盘卸载电机正转3（步）
AND 817.14  ; RK_07 #3托盘下料上升到位感应标志[0017.14]
AND 819.13  ; RK_07 #3托盘下料下降到位感应标志[0019.13]
ANDNOT 117.14  ; RK_07 #3托盘下料电机正转
ANDNOT 117.15  ; RK_07 #3托盘下料电机反转
ORLD
LD D1122.03  ; RK_07 铝壳上料移载机构吸盘破真空3（步）
ANDNOT 117.02  ; RK_07 铝壳上料移载吸盘立真空
ANDNOT 817.02  ; RK_07 铝壳上料移载吸盘真空标志[0017.02]
ANDNOT H50.10  ; RK_07 铝壳上料移载机构吸盘立真空记忆
ANDNOT H51.00  ; RK_07 铝壳上料移载机构有料记忆
ANDNOT H51.10  ; RK_07 铝壳上料移载机构有托盘记忆
AND H66.00  ; RK_07 铝壳托盘下料升降机构有料记忆
ANDNOT 818.01  ; RK_07 #3托盘下料满托盘位（#2）标志[0018.01]
ORLD
LD D1122.04  ; RK_07 铝壳上料移载机构#3铝壳托盘卸载电机反转3（步）
ANDNOT 817.14  ; RK_07 #3托盘下料上升到位感应标志[0017.14]
ANDNOT 819.13  ; RK_07 #3托盘下料下降到位感应标志[0019.13]
ANDNOT 117.14  ; RK_07 #3托盘下料电机正转
ANDNOT 117.15  ; RK_07 #3托盘下料电机反转
AND D1111.00  ; RK_07 铝壳上料移载机构运行条件（公共）
ANDNOT H65.00  ; RK_07 铝壳托盘下料升降机构手动下料记忆
ORLD
LD D1122.05  ; RK_07 铝壳上料移载机构Y轴铝壳取料位&#1/2铝壳上料位3（步）
AND H50.00  ; RK_07 U8_Z 铝壳上料移载Y轴回原点记忆
LDNOT H56.00  ; RK_07 #1铝壳上料升降机构有料记忆
ANDNOT H61.00  ; RK_07 #2铝壳上料升降机构有料记忆
ANDNOT W242.00  ; 铝壳上料移载机构Y轴#1铝壳上料位优先标志
ANDNOT W242.01  ; 铝壳上料移载机构Y轴#2铝壳上料位优先标志
LD 888.00  ; RK_07 U8_Z 铝壳上料移载Y轴#1铝壳取料位标志
ANDNOT 888.01  ; RK_07 U8_Z 铝壳上料移载Y轴#2铝壳取料位标志
LD 888.01  ; RK_07 U8_Z 铝壳上料移载Y轴#2铝壳取料位标志
ANDNOT 888.00  ; RK_07 U8_Z 铝壳上料移载Y轴#1铝壳取料位标志
ORLD
ANDNOT 888.02  ; RK_07 U8_Z 铝壳上料移载Y轴#3铝壳取料位标志
LD 888.02  ; RK_07 U8_Z 铝壳上料移载Y轴#3铝壳取料位标志
ANDNOT 888.00  ; RK_07 U8_Z 铝壳上料移载Y轴#1铝壳取料位标志
ANDNOT 888.01  ; RK_07 U8_Z 铝壳上料移载Y轴#2铝壳取料位标志
ORLD
ANDLD
AND 865.04  ; RK_07 U8_Z 铝壳上料移载Y轴铝壳取料位标志
LD H56.00  ; RK_07 #1铝壳上料升降机构有料记忆
AND W242.00  ; 铝壳上料移载机构Y轴#1铝壳上料位优先标志
AND 865.01  ; RK_07 U8_Z 铝壳上料移载Y轴#1铝壳上料位标志
ORLD
LD H61.00  ; RK_07 #2铝壳上料升降机构有料记忆
AND W242.01  ; 铝壳上料移载机构Y轴#2铝壳上料位优先标志
AND 865.02  ; RK_07 U8_Z 铝壳上料移载Y轴#2铝壳上料位标志
ORLD
ANDLD
ORLD
OR D1122.06  ; 备用
LD D1114.05  ; RK_07 铝壳进料机构单步/自动循环运行中3（铝壳托盘卸载）
AND W1.01  ; 自动模式
@LD D1113.15  ; RK_07 铝壳上料移载机构单步（SW）
AND D1114.12  ; RK_07 铝壳上料移载机构单步运行条件3（铝壳托盘卸载）
ORLD
ANDLD
OUT D1121.01  ; RK_07 铝壳上料移载机构步进条件3（铝壳托盘卸载）

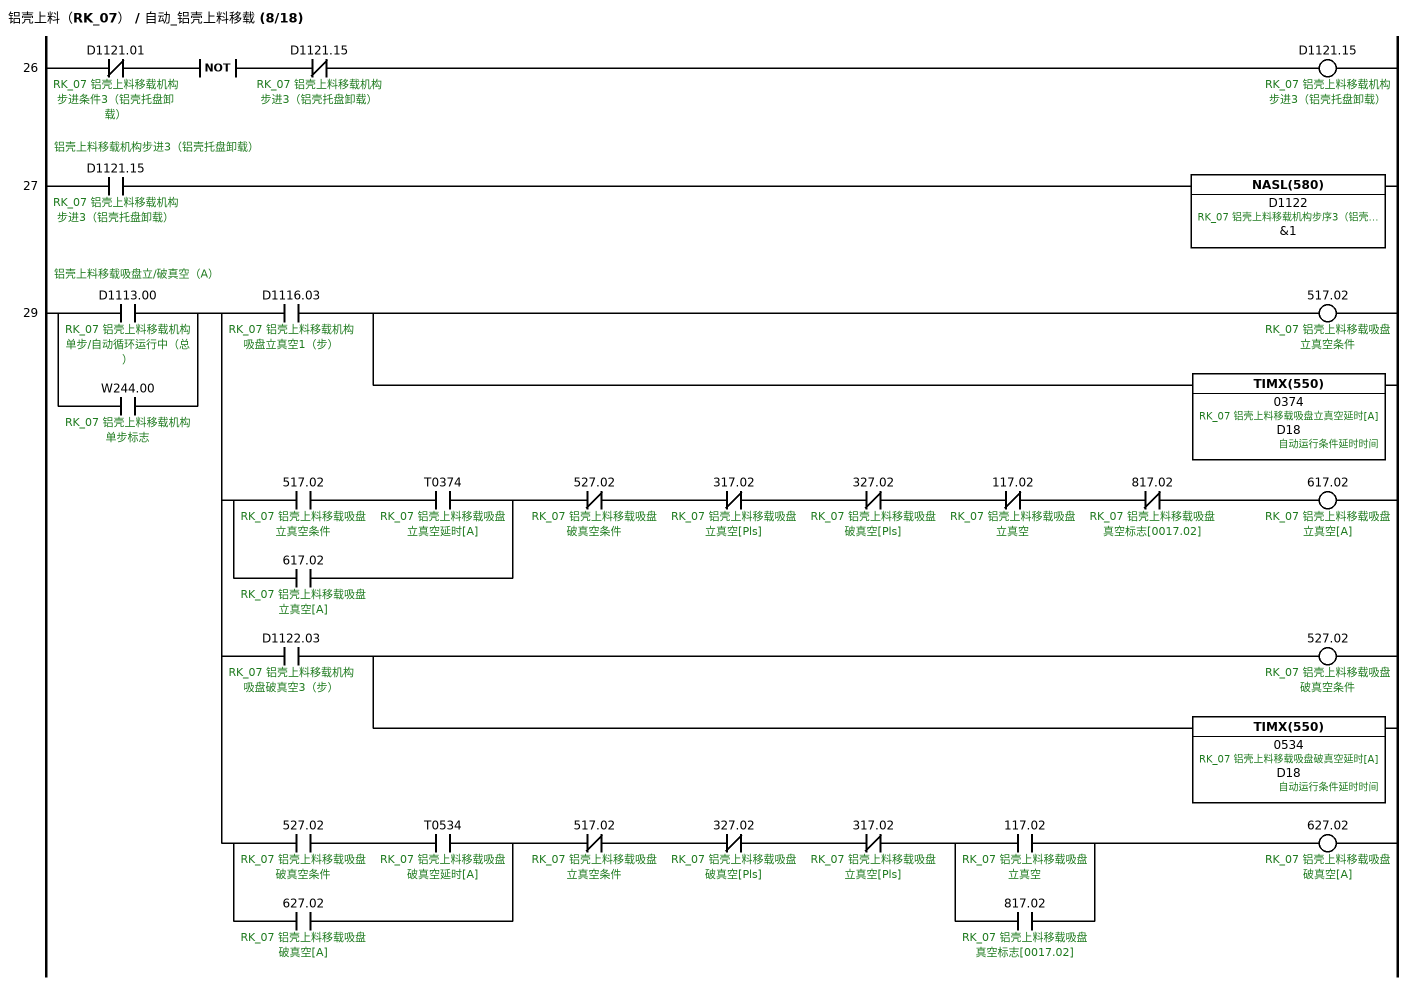
; rung 26
LDNOT D1121.01  ; RK_07 铝壳上料移载机构步进条件3（铝壳托盘卸载）
NOT(520)
ANDNOT D1121.15  ; RK_07 铝壳上料移载机构步进3（铝壳托盘卸载）
OUT D1121.15  ; RK_07 铝壳上料移载机构步进3（铝壳托盘卸载）
; rung 27: 铝壳上料移载机构步进3（铝壳托盘卸载）
LD D1121.15  ; RK_07 铝壳上料移载机构步进3（铝壳托盘卸载）
NASL(580) D1122 &1  ; RK_07 铝壳上料移载机构步序3（铝壳托盘卸载）
; rung 28: 铝壳上料移载机构步序跳转3（铝壳托盘卸载）
; rung 29: 铝壳上料移载吸盘立/破真空（A）
LD D1113.00  ; RK_07 铝壳上料移载机构单步/自动循环运行中（总）
OR W244.00  ; RK_07 铝壳上料移载机构单步标志
OUT TR0
AND D1116.03  ; RK_07 铝壳上料移载机构吸盘立真空1（步）
OUT 517.02  ; RK_07 铝壳上料移载吸盘立真空条件
TIMX(550) 0374 D18  ; 自动运行条件延时时间, RK_07 铝壳上料移载吸盘立真空延时[A]
LD TR0
LD 517.02  ; RK_07 铝壳上料移载吸盘立真空条件
AND T0374  ; RK_07 铝壳上料移载吸盘立真空延时[A]
OR 617.02  ; RK_07 铝壳上料移载吸盘立真空[A]
ANDLD
ANDNOT 527.02  ; RK_07 铝壳上料移载吸盘破真空条件
ANDNOT 317.02  ; RK_07 铝壳上料移载吸盘立真空[Pls]
ANDNOT 327.02  ; RK_07 铝壳上料移载吸盘破真空[Pls]
ANDNOT 117.02  ; RK_07 铝壳上料移载吸盘立真空
ANDNOT 817.02  ; RK_07 铝壳上料移载吸盘真空标志[0017.02]
OUT 617.02  ; RK_07 铝壳上料移载吸盘立真空[A]
LD TR0
AND D1122.03  ; RK_07 铝壳上料移载机构吸盘破真空3（步）
OUT 527.02  ; RK_07 铝壳上料移载吸盘破真空条件
TIMX(550) 0534 D18  ; 自动运行条件延时时间, RK_07 铝壳上料移载吸盘破真空延时[A]
LD TR0
LD 527.02  ; RK_07 铝壳上料移载吸盘破真空条件
AND T0534  ; RK_07 铝壳上料移载吸盘破真空延时[A]
OR 627.02  ; RK_07 铝壳上料移载吸盘破真空[A]
ANDLD
ANDNOT 517.02  ; RK_07 铝壳上料移载吸盘立真空条件
ANDNOT 327.02  ; RK_07 铝壳上料移载吸盘破真空[Pls]
ANDNOT 317.02  ; RK_07 铝壳上料移载吸盘立真空[Pls]
LD 117.02  ; RK_07 铝壳上料移载吸盘立真空
OR 817.02  ; RK_07 铝壳上料移载吸盘真空标志[0017.02]
ANDLD
OUT 627.02  ; RK_07 铝壳上料移载吸盘破真空[A]

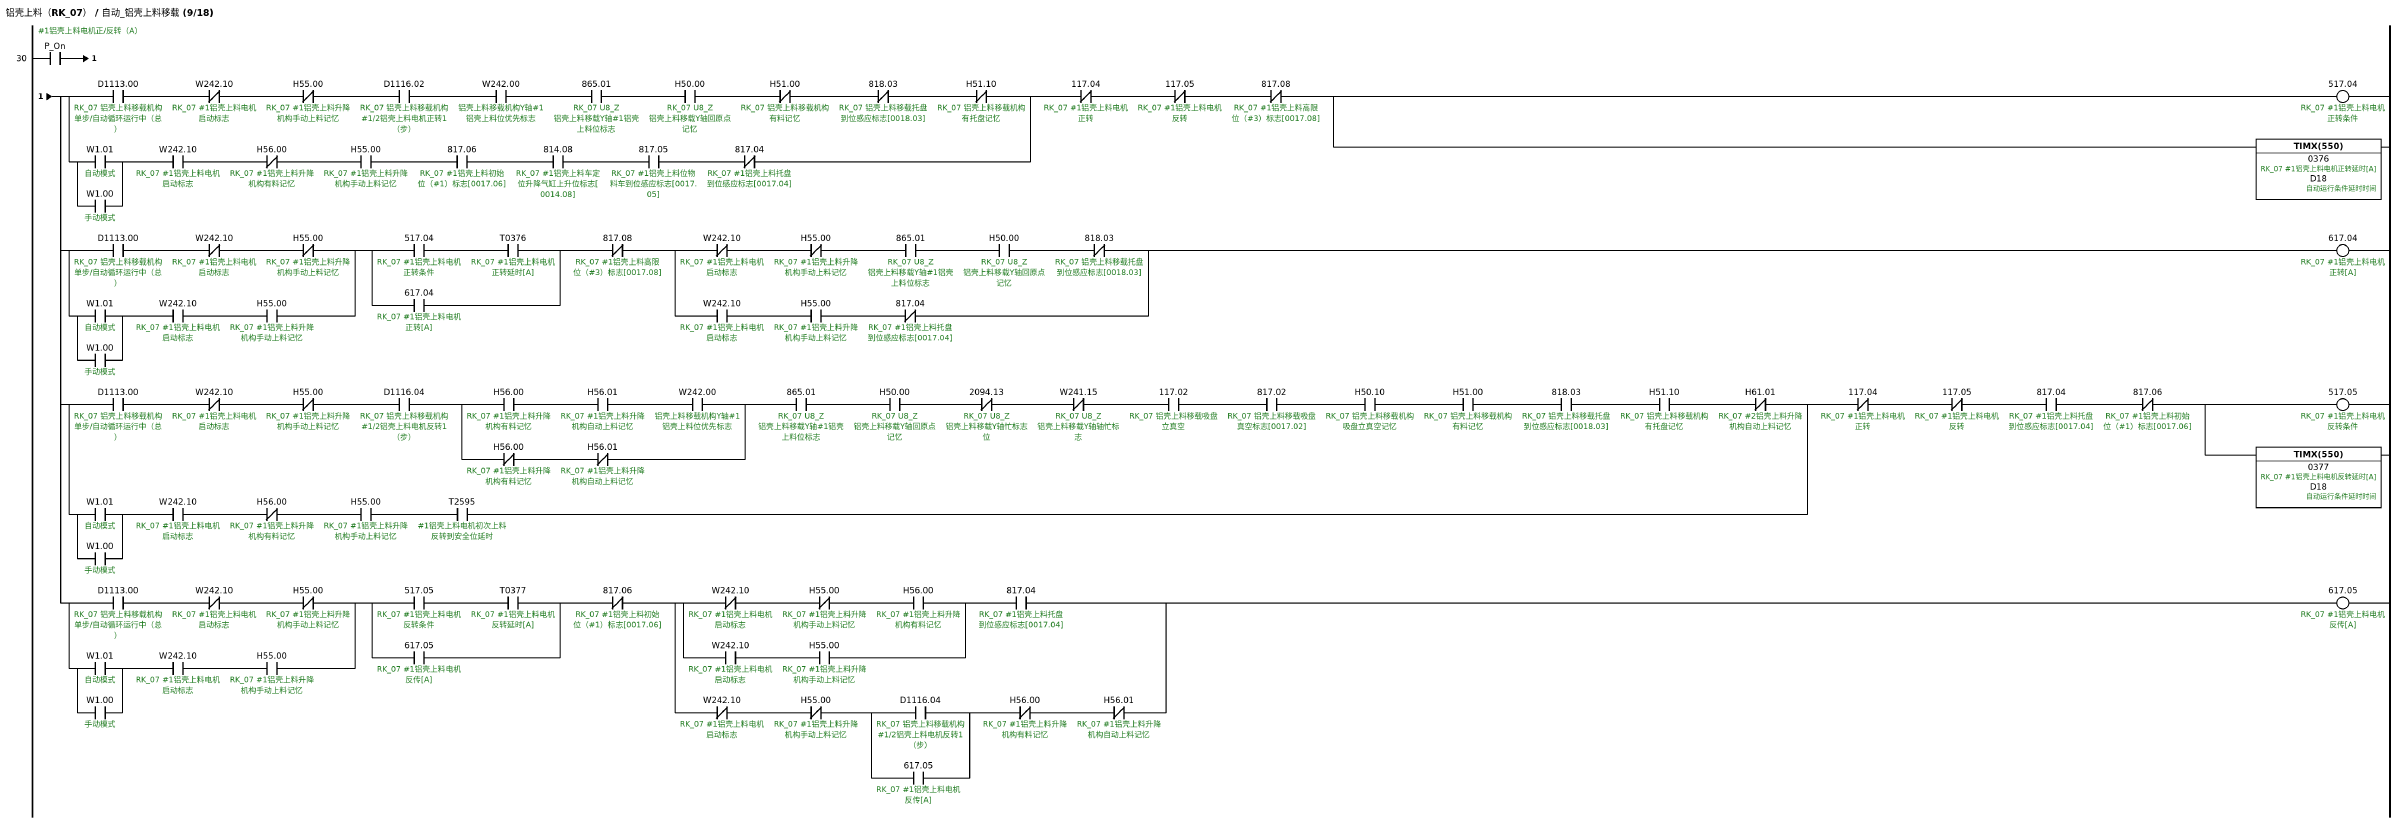
; rung 30: #1铝壳上料电机正/反转（A）
LD P_On
OUT TR0
LD D1113.00  ; RK_07 铝壳上料移载机构单步/自动循环运行中（总）
ANDNOT W242.10  ; RK_07 #1铝壳上料电机启动标志
ANDNOT H55.00  ; RK_07 #1铝壳上料升降机构手动上料记忆
AND D1116.02  ; RK_07 铝壳上料移载机构#1/2铝壳上料电机正转1（步）
AND W242.00  ; 铝壳上料移载机构Y轴#1铝壳上料位优先标志
AND 865.01  ; RK_07 U8_Z 铝壳上料移载Y轴#1铝壳上料位标志
AND H50.00  ; RK_07 U8_Z 铝壳上料移载Y轴回原点记忆
ANDNOT H51.00  ; RK_07 铝壳上料移载机构有料记忆
ANDNOT 818.03  ; RK_07 铝壳上料移载托盘到位感应标志[0018.03]
ANDNOT H51.10  ; RK_07 铝壳上料移载机构有托盘记忆
LD W1.01  ; 自动模式
OR W1.00  ; 手动模式
AND W242.10  ; RK_07 #1铝壳上料电机启动标志
ANDNOT H56.00  ; RK_07 #1铝壳上料升降机构有料记忆
AND H55.00  ; RK_07 #1铝壳上料升降机构手动上料记忆
AND 817.06  ; RK_07 #1铝壳上料初始位（#1）标志[0017.06]
AND 814.08  ; RK_07 #1铝壳上料车定位升降气缸上升位标志[0014.08]
AND 817.05  ; RK_07 #1铝壳上料位物料车到位感应标志[0017.05]
ANDNOT 817.04  ; RK_07 #1铝壳上料托盘到位感应标志[0017.04]
ORLD
ANDLD
ANDNOT 117.04  ; RK_07 #1铝壳上料电机正转
ANDNOT 117.05  ; RK_07 #1铝壳上料电机反转
ANDNOT 817.08  ; RK_07 #1铝壳上料高限位（#3）标志[0017.08]
OUT 517.04  ; RK_07 #1铝壳上料电机正转条件
TIMX(550) 0376 D18  ; 自动运行条件延时时间, RK_07 #1铝壳上料电机正转延时[A]
LD TR0
LD D1113.00  ; RK_07 铝壳上料移载机构单步/自动循环运行中（总）
ANDNOT W242.10  ; RK_07 #1铝壳上料电机启动标志
ANDNOT H55.00  ; RK_07 #1铝壳上料升降机构手动上料记忆
LD W1.01  ; 自动模式
OR W1.00  ; 手动模式
AND W242.10  ; RK_07 #1铝壳上料电机启动标志
AND H55.00  ; RK_07 #1铝壳上料升降机构手动上料记忆
ORLD
ANDLD
LD 517.04  ; RK_07 #1铝壳上料电机正转条件
AND T0376  ; RK_07 #1铝壳上料电机正转延时[A]
OR 617.04  ; RK_07 #1铝壳上料电机正转[A]
ANDLD
ANDNOT 817.08  ; RK_07 #1铝壳上料高限位（#3）标志[0017.08]
LDNOT W242.10  ; RK_07 #1铝壳上料电机启动标志
ANDNOT H55.00  ; RK_07 #1铝壳上料升降机构手动上料记忆
AND 865.01  ; RK_07 U8_Z 铝壳上料移载Y轴#1铝壳上料位标志
AND H50.00  ; RK_07 U8_Z 铝壳上料移载Y轴回原点记忆
ANDNOT 818.03  ; RK_07 铝壳上料移载托盘到位感应标志[0018.03]
LD W242.10  ; RK_07 #1铝壳上料电机启动标志
AND H55.00  ; RK_07 #1铝壳上料升降机构手动上料记忆
ANDNOT 817.04  ; RK_07 #1铝壳上料托盘到位感应标志[0017.04]
ORLD
ANDLD
OUT 617.04  ; RK_07 #1铝壳上料电机正转[A]
LD TR0
LD D1113.00  ; RK_07 铝壳上料移载机构单步/自动循环运行中（总）
ANDNOT W242.10  ; RK_07 #1铝壳上料电机启动标志
ANDNOT H55.00  ; RK_07 #1铝壳上料升降机构手动上料记忆
AND D1116.04  ; RK_07 铝壳上料移载机构#1/2铝壳上料电机反转1（步）
LD H56.00  ; RK_07 #1铝壳上料升降机构有料记忆
AND H56.01  ; RK_07 #1铝壳上料升降机构自动上料记忆
AND W242.00  ; 铝壳上料移载机构Y轴#1铝壳上料位优先标志
LDNOT H56.00  ; RK_07 #1铝壳上料升降机构有料记忆
ANDNOT H56.01  ; RK_07 #1铝壳上料升降机构自动上料记忆
ORLD
ANDLD
AND 865.01  ; RK_07 U8_Z 铝壳上料移载Y轴#1铝壳上料位标志
AND H50.00  ; RK_07 U8_Z 铝壳上料移载Y轴回原点记忆
ANDNOT 2094.13  ; RK_07 U8_Z 铝壳上料移载Y轴忙标志位
ANDNOT W241.15  ; RK_07 U8_Z 铝壳上料移载Y轴轴忙标志
AND 117.02  ; RK_07 铝壳上料移载吸盘立真空
AND 817.02  ; RK_07 铝壳上料移载吸盘真空标志[0017.02]
AND H50.10  ; RK_07 铝壳上料移载机构吸盘立真空记忆
AND H51.00  ; RK_07 铝壳上料移载机构有料记忆
AND 818.03  ; RK_07 铝壳上料移载托盘到位感应标志[0018.03]
AND H51.10  ; RK_07 铝壳上料移载机构有托盘记忆
ANDNOT H61.01  ; RK_07 #2铝壳上料升降机构自动上料记忆
LD W1.01  ; 自动模式
OR W1.00  ; 手动模式
AND W242.10  ; RK_07 #1铝壳上料电机启动标志
ANDNOT H56.00  ; RK_07 #1铝壳上料升降机构有料记忆
AND H55.00  ; RK_07 #1铝壳上料升降机构手动上料记忆
AND T2595  ; #1铝壳上料电机初次上料反转到安全位延时
ORLD
ANDLD
ANDNOT 117.04  ; RK_07 #1铝壳上料电机正转
ANDNOT 117.05  ; RK_07 #1铝壳上料电机反转
AND 817.04  ; RK_07 #1铝壳上料托盘到位感应标志[0017.04]
ANDNOT 817.06  ; RK_07 #1铝壳上料初始位（#1）标志[0017.06]
OUT 517.05  ; RK_07 #1铝壳上料电机反转条件
TIMX(550) 0377 D18  ; 自动运行条件延时时间, RK_07 #1铝壳上料电机反转延时[A]
LD TR0
LD D1113.00  ; RK_07 铝壳上料移载机构单步/自动循环运行中（总）
ANDNOT W242.10  ; RK_07 #1铝壳上料电机启动标志
ANDNOT H55.00  ; RK_07 #1铝壳上料升降机构手动上料记忆
LD W1.01  ; 自动模式
OR W1.00  ; 手动模式
AND W242.10  ; RK_07 #1铝壳上料电机启动标志
AND H55.00  ; RK_07 #1铝壳上料升降机构手动上料记忆
ORLD
ANDLD
LD 517.05  ; RK_07 #1铝壳上料电机反转条件
AND T0377  ; RK_07 #1铝壳上料电机反转延时[A]
OR 617.05  ; RK_07 #1铝壳上料电机反传[A]
ANDLD
ANDNOT 817.06  ; RK_07 #1铝壳上料初始位（#1）标志[0017.06]
LDNOT W242.10  ; RK_07 #1铝壳上料电机启动标志
ANDNOT H55.00  ; RK_07 #1铝壳上料升降机构手动上料记忆
AND H56.00  ; RK_07 #1铝壳上料升降机构有料记忆
LD W242.10  ; RK_07 #1铝壳上料电机启动标志
AND H55.00  ; RK_07 #1铝壳上料升降机构手动上料记忆
ORLD
AND 817.04  ; RK_07 #1铝壳上料托盘到位感应标志[0017.04]
LDNOT W242.10  ; RK_07 #1铝壳上料电机启动标志
ANDNOT H55.00  ; RK_07 #1铝壳上料升降机构手动上料记忆
LD D1116.04  ; RK_07 铝壳上料移载机构#1/2铝壳上料电机反转1（步）
OR 617.05  ; RK_07 #1铝壳上料电机反传[A]
ANDLD
ANDNOT H56.00  ; RK_07 #1铝壳上料升降机构有料记忆
ANDNOT H56.01  ; RK_07 #1铝壳上料升降机构自动上料记忆
ORLD
ANDLD
OUT 617.05  ; RK_07 #1铝壳上料电机反传[A]

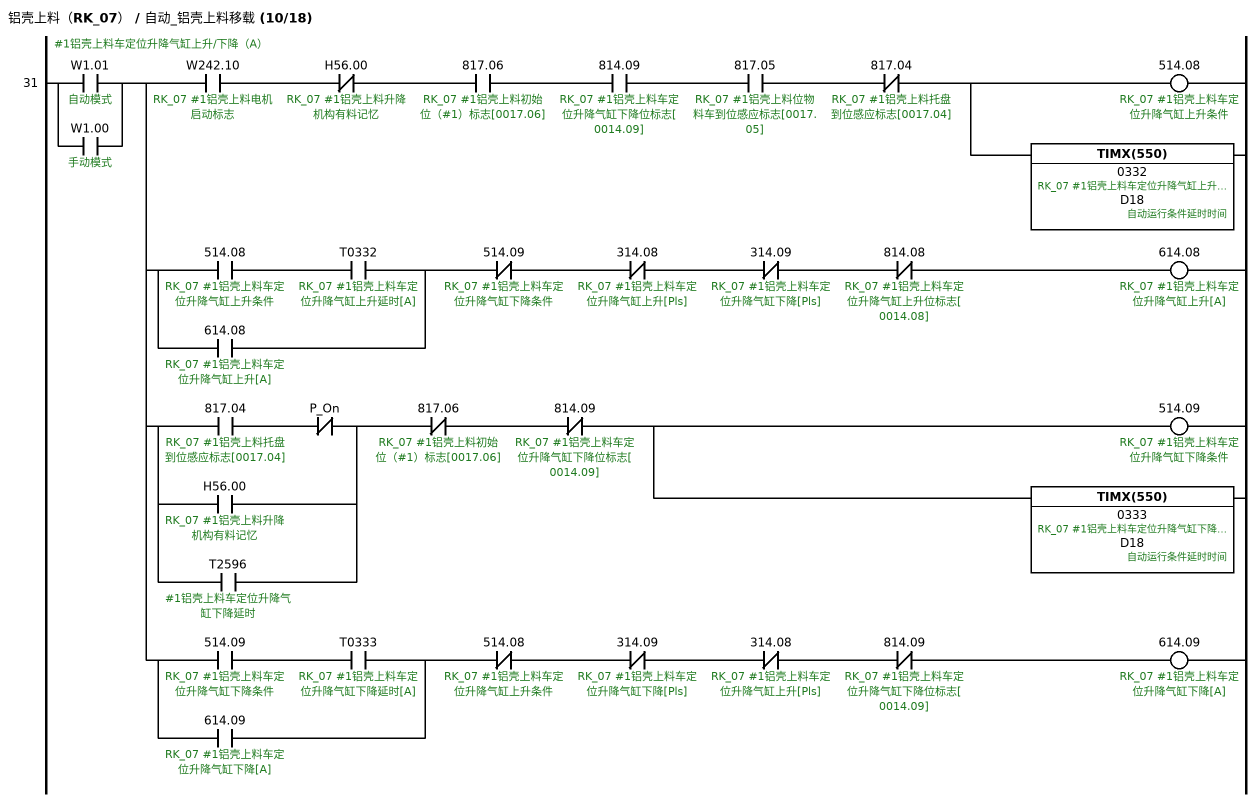
; rung 31: #1铝壳上料车定位升降气缸上升/下降（A）
LD W1.01  ; 自动模式
OR W1.00  ; 手动模式
OUT TR0
AND W242.10  ; RK_07 #1铝壳上料电机启动标志
ANDNOT H56.00  ; RK_07 #1铝壳上料升降机构有料记忆
AND 817.06  ; RK_07 #1铝壳上料初始位（#1）标志[0017.06]
AND 814.09  ; RK_07 #1铝壳上料车定位升降气缸下降位标志[0014.09]
AND 817.05  ; RK_07 #1铝壳上料位物料车到位感应标志[0017.05]
ANDNOT 817.04  ; RK_07 #1铝壳上料托盘到位感应标志[0017.04]
OUT 514.08  ; RK_07 #1铝壳上料车定位升降气缸上升条件
TIMX(550) 0332 D18  ; 自动运行条件延时时间, RK_07 #1铝壳上料车定位升降气缸上升延时[A]
LD TR0
LD 514.08  ; RK_07 #1铝壳上料车定位升降气缸上升条件
AND T0332  ; RK_07 #1铝壳上料车定位升降气缸上升延时[A]
OR 614.08  ; RK_07 #1铝壳上料车定位升降气缸上升[A]
ANDLD
ANDNOT 514.09  ; RK_07 #1铝壳上料车定位升降气缸下降条件
ANDNOT 314.08  ; RK_07 #1铝壳上料车定位升降气缸上升[Pls]
ANDNOT 314.09  ; RK_07 #1铝壳上料车定位升降气缸下降[Pls]
ANDNOT 814.08  ; RK_07 #1铝壳上料车定位升降气缸上升位标志[0014.08]
OUT 614.08  ; RK_07 #1铝壳上料车定位升降气缸上升[A]
LD TR0
LD 817.04  ; RK_07 #1铝壳上料托盘到位感应标志[0017.04]
ANDNOT P_On
OR H56.00  ; RK_07 #1铝壳上料升降机构有料记忆
OR T2596  ; #1铝壳上料车定位升降气缸下降延时
ANDLD
ANDNOT 817.06  ; RK_07 #1铝壳上料初始位（#1）标志[0017.06]
ANDNOT 814.09  ; RK_07 #1铝壳上料车定位升降气缸下降位标志[0014.09]
OUT 514.09  ; RK_07 #1铝壳上料车定位升降气缸下降条件
TIMX(550) 0333 D18  ; 自动运行条件延时时间, RK_07 #1铝壳上料车定位升降气缸下降延时[A]
LD TR0
LD 514.09  ; RK_07 #1铝壳上料车定位升降气缸下降条件
AND T0333  ; RK_07 #1铝壳上料车定位升降气缸下降延时[A]
OR 614.09  ; RK_07 #1铝壳上料车定位升降气缸下降[A]
ANDLD
ANDNOT 514.08  ; RK_07 #1铝壳上料车定位升降气缸上升条件
ANDNOT 314.09  ; RK_07 #1铝壳上料车定位升降气缸下降[Pls]
ANDNOT 314.08  ; RK_07 #1铝壳上料车定位升降气缸上升[Pls]
ANDNOT 814.09  ; RK_07 #1铝壳上料车定位升降气缸下降位标志[0014.09]
OUT 614.09  ; RK_07 #1铝壳上料车定位升降气缸下降[A]

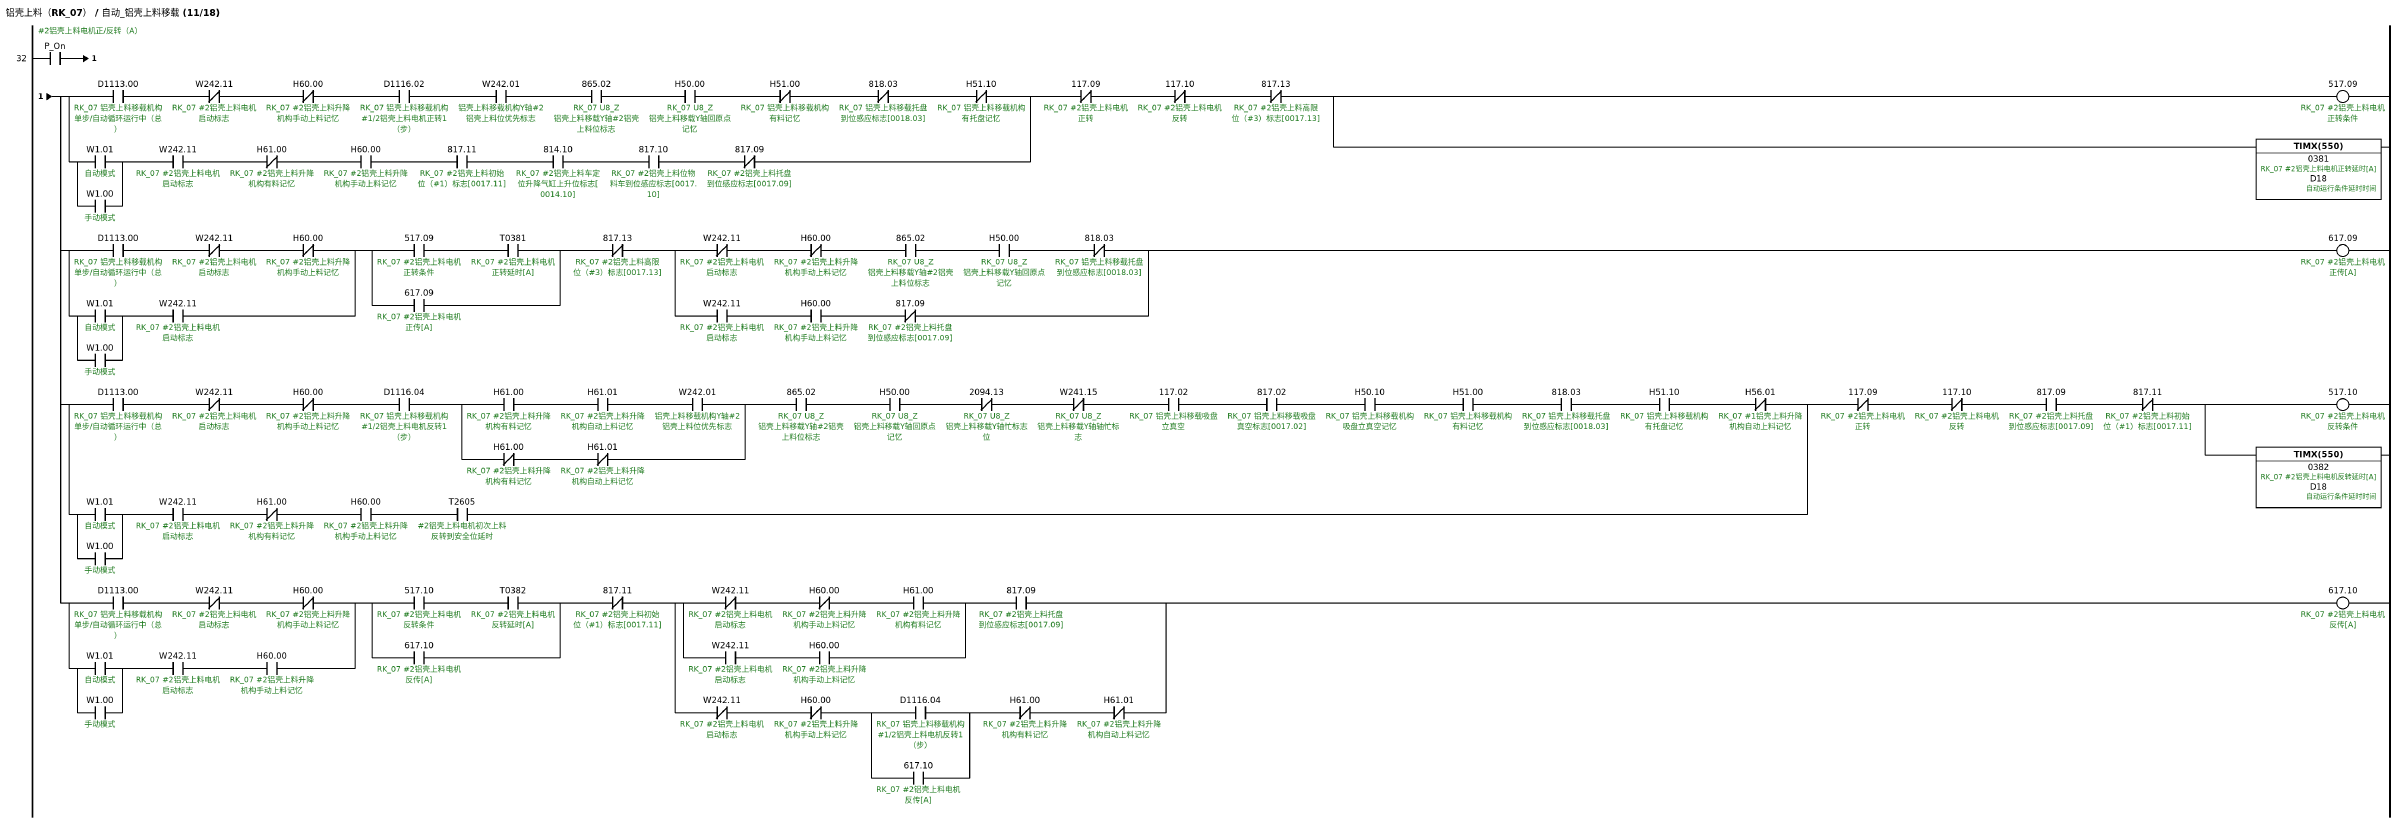
; rung 32: #2铝壳上料电机正/反转（A）
LD P_On
OUT TR0
LD D1113.00  ; RK_07 铝壳上料移载机构单步/自动循环运行中（总）
ANDNOT W242.11  ; RK_07 #2铝壳上料电机启动标志
ANDNOT H60.00  ; RK_07 #2铝壳上料升降机构手动上料记忆
AND D1116.02  ; RK_07 铝壳上料移载机构#1/2铝壳上料电机正转1（步）
AND W242.01  ; 铝壳上料移载机构Y轴#2铝壳上料位优先标志
AND 865.02  ; RK_07 U8_Z 铝壳上料移载Y轴#2铝壳上料位标志
AND H50.00  ; RK_07 U8_Z 铝壳上料移载Y轴回原点记忆
ANDNOT H51.00  ; RK_07 铝壳上料移载机构有料记忆
ANDNOT 818.03  ; RK_07 铝壳上料移载托盘到位感应标志[0018.03]
ANDNOT H51.10  ; RK_07 铝壳上料移载机构有托盘记忆
LD W1.01  ; 自动模式
OR W1.00  ; 手动模式
AND W242.11  ; RK_07 #2铝壳上料电机启动标志
ANDNOT H61.00  ; RK_07 #2铝壳上料升降机构有料记忆
AND H60.00  ; RK_07 #2铝壳上料升降机构手动上料记忆
AND 817.11  ; RK_07 #2铝壳上料初始位（#1）标志[0017.11]
AND 814.10  ; RK_07 #2铝壳上料车定位升降气缸上升位标志[0014.10]
AND 817.10  ; RK_07 #2铝壳上料位物料车到位感应标志[0017.10]
ANDNOT 817.09  ; RK_07 #2铝壳上料托盘到位感应标志[0017.09]
ORLD
ANDLD
ANDNOT 117.09  ; RK_07 #2铝壳上料电机正转
ANDNOT 117.10  ; RK_07 #2铝壳上料电机反转
ANDNOT 817.13  ; RK_07 #2铝壳上料高限位（#3）标志[0017.13]
OUT 517.09  ; RK_07 #2铝壳上料电机正转条件
TIMX(550) 0381 D18  ; 自动运行条件延时时间, RK_07 #2铝壳上料电机正转延时[A]
LD TR0
LD D1113.00  ; RK_07 铝壳上料移载机构单步/自动循环运行中（总）
ANDNOT W242.11  ; RK_07 #2铝壳上料电机启动标志
ANDNOT H60.00  ; RK_07 #2铝壳上料升降机构手动上料记忆
LD W1.01  ; 自动模式
OR W1.00  ; 手动模式
AND W242.11  ; RK_07 #2铝壳上料电机启动标志
ORLD
ANDLD
LD 517.09  ; RK_07 #2铝壳上料电机正转条件
AND T0381  ; RK_07 #2铝壳上料电机正转延时[A]
OR 617.09  ; RK_07 #2铝壳上料电机正传[A]
ANDLD
ANDNOT 817.13  ; RK_07 #2铝壳上料高限位（#3）标志[0017.13]
LDNOT W242.11  ; RK_07 #2铝壳上料电机启动标志
ANDNOT H60.00  ; RK_07 #2铝壳上料升降机构手动上料记忆
AND 865.02  ; RK_07 U8_Z 铝壳上料移载Y轴#2铝壳上料位标志
AND H50.00  ; RK_07 U8_Z 铝壳上料移载Y轴回原点记忆
ANDNOT 818.03  ; RK_07 铝壳上料移载托盘到位感应标志[0018.03]
LD W242.11  ; RK_07 #2铝壳上料电机启动标志
AND H60.00  ; RK_07 #2铝壳上料升降机构手动上料记忆
ANDNOT 817.09  ; RK_07 #2铝壳上料托盘到位感应标志[0017.09]
ORLD
ANDLD
OUT 617.09  ; RK_07 #2铝壳上料电机正传[A]
LD TR0
LD D1113.00  ; RK_07 铝壳上料移载机构单步/自动循环运行中（总）
ANDNOT W242.11  ; RK_07 #2铝壳上料电机启动标志
ANDNOT H60.00  ; RK_07 #2铝壳上料升降机构手动上料记忆
AND D1116.04  ; RK_07 铝壳上料移载机构#1/2铝壳上料电机反转1（步）
LD H61.00  ; RK_07 #2铝壳上料升降机构有料记忆
AND H61.01  ; RK_07 #2铝壳上料升降机构自动上料记忆
AND W242.01  ; 铝壳上料移载机构Y轴#2铝壳上料位优先标志
LDNOT H61.00  ; RK_07 #2铝壳上料升降机构有料记忆
ANDNOT H61.01  ; RK_07 #2铝壳上料升降机构自动上料记忆
ORLD
ANDLD
AND 865.02  ; RK_07 U8_Z 铝壳上料移载Y轴#2铝壳上料位标志
AND H50.00  ; RK_07 U8_Z 铝壳上料移载Y轴回原点记忆
ANDNOT 2094.13  ; RK_07 U8_Z 铝壳上料移载Y轴忙标志位
ANDNOT W241.15  ; RK_07 U8_Z 铝壳上料移载Y轴轴忙标志
AND 117.02  ; RK_07 铝壳上料移载吸盘立真空
AND 817.02  ; RK_07 铝壳上料移载吸盘真空标志[0017.02]
AND H50.10  ; RK_07 铝壳上料移载机构吸盘立真空记忆
AND H51.00  ; RK_07 铝壳上料移载机构有料记忆
AND 818.03  ; RK_07 铝壳上料移载托盘到位感应标志[0018.03]
AND H51.10  ; RK_07 铝壳上料移载机构有托盘记忆
ANDNOT H56.01  ; RK_07 #1铝壳上料升降机构自动上料记忆
LD W1.01  ; 自动模式
OR W1.00  ; 手动模式
AND W242.11  ; RK_07 #2铝壳上料电机启动标志
ANDNOT H61.00  ; RK_07 #2铝壳上料升降机构有料记忆
AND H60.00  ; RK_07 #2铝壳上料升降机构手动上料记忆
AND T2605  ; #2铝壳上料电机初次上料反转到安全位延时
ORLD
ANDLD
ANDNOT 117.09  ; RK_07 #2铝壳上料电机正转
ANDNOT 117.10  ; RK_07 #2铝壳上料电机反转
AND 817.09  ; RK_07 #2铝壳上料托盘到位感应标志[0017.09]
ANDNOT 817.11  ; RK_07 #2铝壳上料初始位（#1）标志[0017.11]
OUT 517.10  ; RK_07 #2铝壳上料电机反转条件
TIMX(550) 0382 D18  ; 自动运行条件延时时间, RK_07 #2铝壳上料电机反转延时[A]
LD TR0
LD D1113.00  ; RK_07 铝壳上料移载机构单步/自动循环运行中（总）
ANDNOT W242.11  ; RK_07 #2铝壳上料电机启动标志
ANDNOT H60.00  ; RK_07 #2铝壳上料升降机构手动上料记忆
LD W1.01  ; 自动模式
OR W1.00  ; 手动模式
AND W242.11  ; RK_07 #2铝壳上料电机启动标志
AND H60.00  ; RK_07 #2铝壳上料升降机构手动上料记忆
ORLD
ANDLD
LD 517.10  ; RK_07 #2铝壳上料电机反转条件
AND T0382  ; RK_07 #2铝壳上料电机反转延时[A]
OR 617.10  ; RK_07 #2铝壳上料电机反传[A]
ANDLD
ANDNOT 817.11  ; RK_07 #2铝壳上料初始位（#1）标志[0017.11]
LDNOT W242.11  ; RK_07 #2铝壳上料电机启动标志
ANDNOT H60.00  ; RK_07 #2铝壳上料升降机构手动上料记忆
AND H61.00  ; RK_07 #2铝壳上料升降机构有料记忆
LD W242.11  ; RK_07 #2铝壳上料电机启动标志
AND H60.00  ; RK_07 #2铝壳上料升降机构手动上料记忆
ORLD
AND 817.09  ; RK_07 #2铝壳上料托盘到位感应标志[0017.09]
LDNOT W242.11  ; RK_07 #2铝壳上料电机启动标志
ANDNOT H60.00  ; RK_07 #2铝壳上料升降机构手动上料记忆
LD D1116.04  ; RK_07 铝壳上料移载机构#1/2铝壳上料电机反转1（步）
OR 617.10  ; RK_07 #2铝壳上料电机反传[A]
ANDLD
ANDNOT H61.00  ; RK_07 #2铝壳上料升降机构有料记忆
ANDNOT H61.01  ; RK_07 #2铝壳上料升降机构自动上料记忆
ORLD
ANDLD
OUT 617.10  ; RK_07 #2铝壳上料电机反传[A]

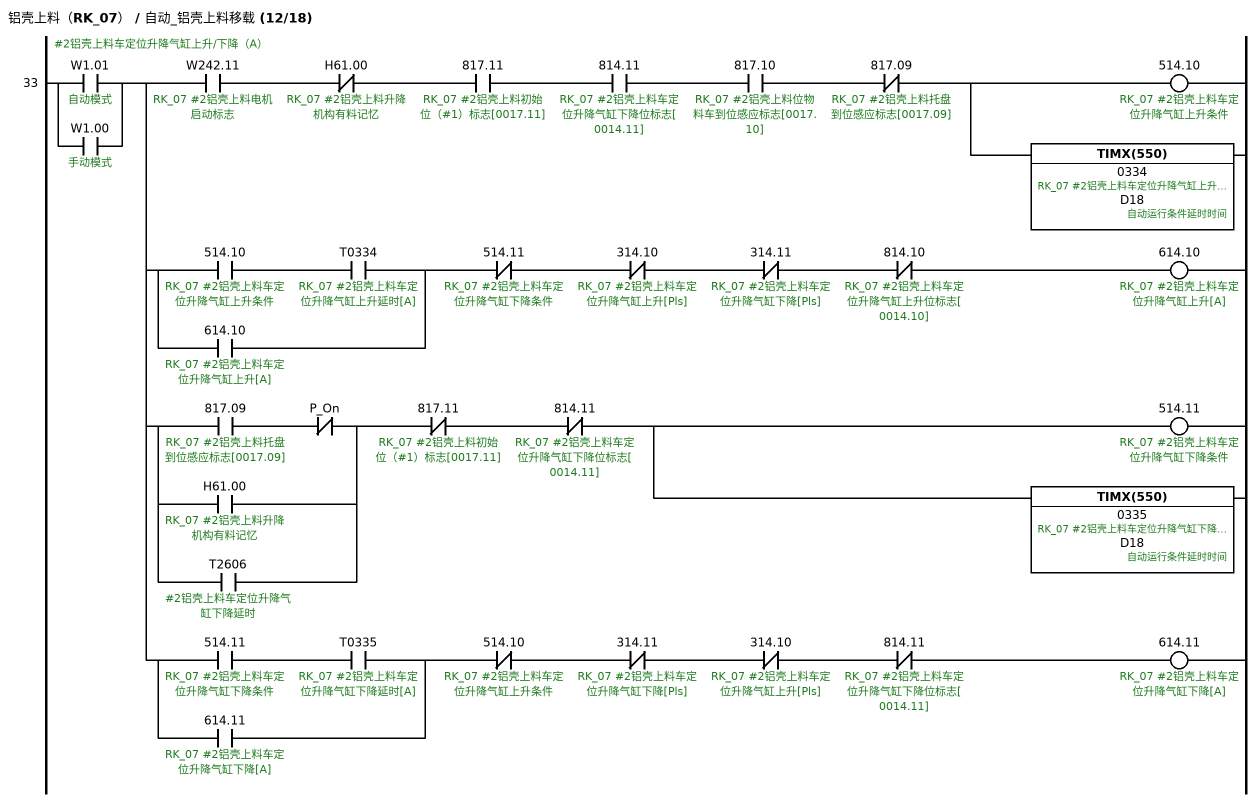
; rung 33: #2铝壳上料车定位升降气缸上升/下降（A）
LD W1.01  ; 自动模式
OR W1.00  ; 手动模式
OUT TR0
AND W242.11  ; RK_07 #2铝壳上料电机启动标志
ANDNOT H61.00  ; RK_07 #2铝壳上料升降机构有料记忆
AND 817.11  ; RK_07 #2铝壳上料初始位（#1）标志[0017.11]
AND 814.11  ; RK_07 #2铝壳上料车定位升降气缸下降位标志[0014.11]
AND 817.10  ; RK_07 #2铝壳上料位物料车到位感应标志[0017.10]
ANDNOT 817.09  ; RK_07 #2铝壳上料托盘到位感应标志[0017.09]
OUT 514.10  ; RK_07 #2铝壳上料车定位升降气缸上升条件
TIMX(550) 0334 D18  ; 自动运行条件延时时间, RK_07 #2铝壳上料车定位升降气缸上升延时[A]
LD TR0
LD 514.10  ; RK_07 #2铝壳上料车定位升降气缸上升条件
AND T0334  ; RK_07 #2铝壳上料车定位升降气缸上升延时[A]
OR 614.10  ; RK_07 #2铝壳上料车定位升降气缸上升[A]
ANDLD
ANDNOT 514.11  ; RK_07 #2铝壳上料车定位升降气缸下降条件
ANDNOT 314.10  ; RK_07 #2铝壳上料车定位升降气缸上升[Pls]
ANDNOT 314.11  ; RK_07 #2铝壳上料车定位升降气缸下降[Pls]
ANDNOT 814.10  ; RK_07 #2铝壳上料车定位升降气缸上升位标志[0014.10]
OUT 614.10  ; RK_07 #2铝壳上料车定位升降气缸上升[A]
LD TR0
LD 817.09  ; RK_07 #2铝壳上料托盘到位感应标志[0017.09]
ANDNOT P_On
OR H61.00  ; RK_07 #2铝壳上料升降机构有料记忆
OR T2606  ; #2铝壳上料车定位升降气缸下降延时
ANDLD
ANDNOT 817.11  ; RK_07 #2铝壳上料初始位（#1）标志[0017.11]
ANDNOT 814.11  ; RK_07 #2铝壳上料车定位升降气缸下降位标志[0014.11]
OUT 514.11  ; RK_07 #2铝壳上料车定位升降气缸下降条件
TIMX(550) 0335 D18  ; 自动运行条件延时时间, RK_07 #2铝壳上料车定位升降气缸下降延时[A]
LD TR0
LD 514.11  ; RK_07 #2铝壳上料车定位升降气缸下降条件
AND T0335  ; RK_07 #2铝壳上料车定位升降气缸下降延时[A]
OR 614.11  ; RK_07 #2铝壳上料车定位升降气缸下降[A]
ANDLD
ANDNOT 514.10  ; RK_07 #2铝壳上料车定位升降气缸上升条件
ANDNOT 314.11  ; RK_07 #2铝壳上料车定位升降气缸下降[Pls]
ANDNOT 314.10  ; RK_07 #2铝壳上料车定位升降气缸上升[Pls]
ANDNOT 814.11  ; RK_07 #2铝壳上料车定位升降气缸下降位标志[0014.11]
OUT 614.11  ; RK_07 #2铝壳上料车定位升降气缸下降[A]

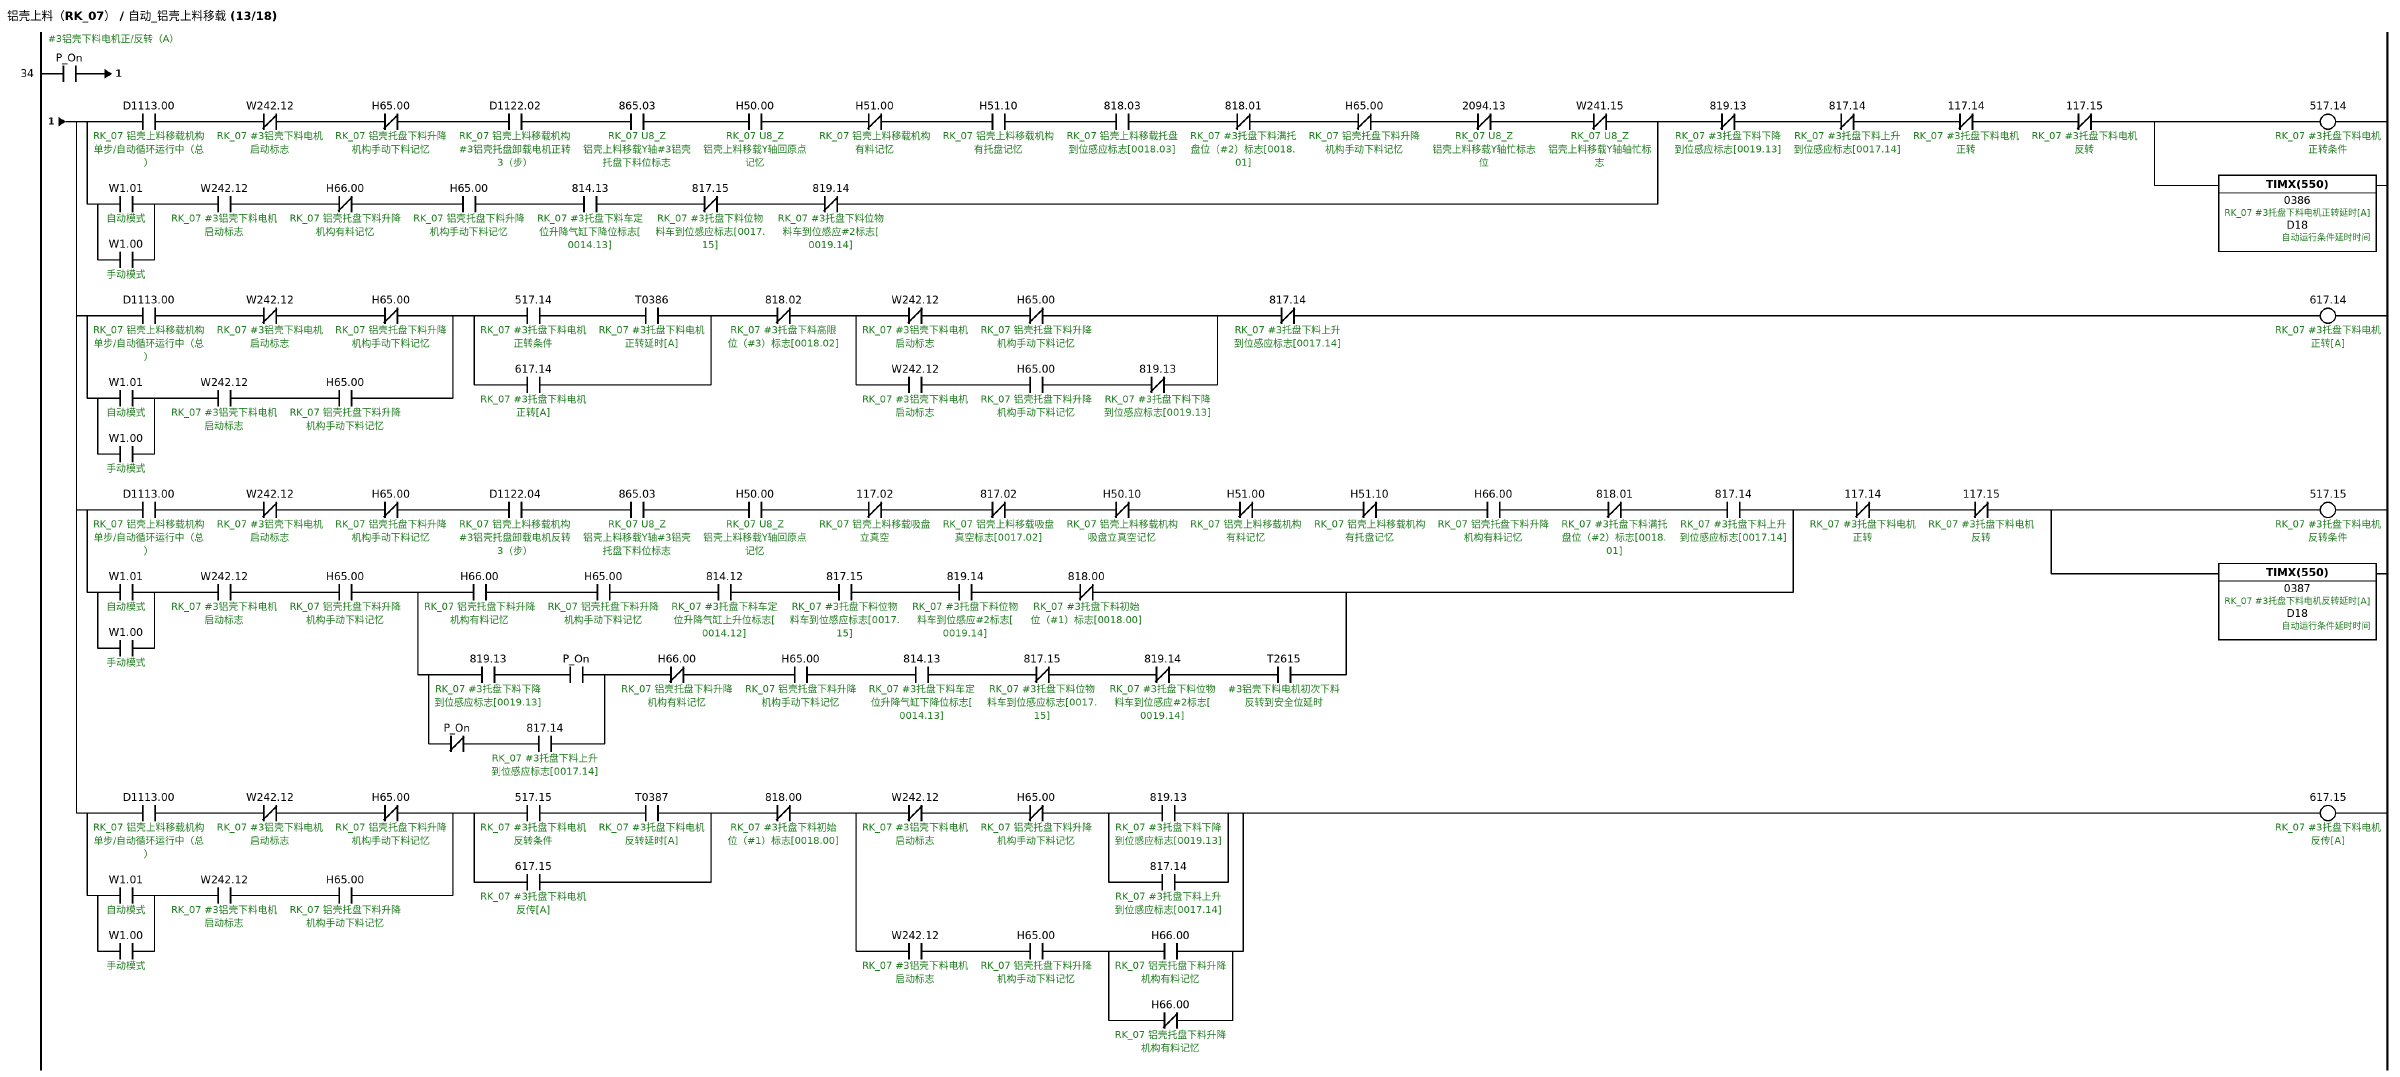
; rung 34: #3铝壳下料电机正/反转（A）
LD P_On
OUT TR0
LD D1113.00  ; RK_07 铝壳上料移载机构单步/自动循环运行中（总）
ANDNOT W242.12  ; RK_07 #3铝壳下料电机启动标志
ANDNOT H65.00  ; RK_07 铝壳托盘下料升降机构手动下料记忆
AND D1122.02  ; RK_07 铝壳上料移载机构#3铝壳托盘卸载电机正转3（步）
AND 865.03  ; RK_07 U8_Z 铝壳上料移载Y轴#3铝壳托盘下料位标志
AND H50.00  ; RK_07 U8_Z 铝壳上料移载Y轴回原点记忆
ANDNOT H51.00  ; RK_07 铝壳上料移载机构有料记忆
AND H51.10  ; RK_07 铝壳上料移载机构有托盘记忆
AND 818.03  ; RK_07 铝壳上料移载托盘到位感应标志[0018.03]
ANDNOT 818.01  ; RK_07 #3托盘下料满托盘位（#2）标志[0018.01]
ANDNOT H65.00  ; RK_07 铝壳托盘下料升降机构手动下料记忆
ANDNOT 2094.13  ; RK_07 U8_Z 铝壳上料移载Y轴忙标志位
ANDNOT W241.15  ; RK_07 U8_Z 铝壳上料移载Y轴轴忙标志
LD W1.01  ; 自动模式
OR W1.00  ; 手动模式
AND W242.12  ; RK_07 #3铝壳下料电机启动标志
ANDNOT H66.00  ; RK_07 铝壳托盘下料升降机构有料记忆
AND H65.00  ; RK_07 铝壳托盘下料升降机构手动下料记忆
AND 814.13  ; RK_07 #3托盘下料车定位升降气缸下降位标志[0014.13]
ANDNOT 817.15  ; RK_07 #3托盘下料位物料车到位感应标志[0017.15]
ANDNOT 819.14  ; RK_07 #3托盘下料位物料车到位感应#2标志[0019.14]
ORLD
ANDLD
ANDNOT 819.13  ; RK_07 #3托盘下料下降到位感应标志[0019.13]
ANDNOT 817.14  ; RK_07 #3托盘下料上升到位感应标志[0017.14]
ANDNOT 117.14  ; RK_07 #3托盘下料电机正转
ANDNOT 117.15  ; RK_07 #3托盘下料电机反转
OUT 517.14  ; RK_07 #3托盘下料电机正转条件
TIMX(550) 0386 D18  ; 自动运行条件延时时间, RK_07 #3托盘下料电机正转延时[A]
LD TR0
LD D1113.00  ; RK_07 铝壳上料移载机构单步/自动循环运行中（总）
ANDNOT W242.12  ; RK_07 #3铝壳下料电机启动标志
ANDNOT H65.00  ; RK_07 铝壳托盘下料升降机构手动下料记忆
LD W1.01  ; 自动模式
OR W1.00  ; 手动模式
AND W242.12  ; RK_07 #3铝壳下料电机启动标志
AND H65.00  ; RK_07 铝壳托盘下料升降机构手动下料记忆
ORLD
ANDLD
LD 517.14  ; RK_07 #3托盘下料电机正转条件
AND T0386  ; RK_07 #3托盘下料电机正转延时[A]
OR 617.14  ; RK_07 #3托盘下料电机正转[A]
ANDLD
ANDNOT 818.02  ; RK_07 #3托盘下料高限位（#3）标志[0018.02]
LDNOT W242.12  ; RK_07 #3铝壳下料电机启动标志
ANDNOT H65.00  ; RK_07 铝壳托盘下料升降机构手动下料记忆
LD W242.12  ; RK_07 #3铝壳下料电机启动标志
AND H65.00  ; RK_07 铝壳托盘下料升降机构手动下料记忆
ANDNOT 819.13  ; RK_07 #3托盘下料下降到位感应标志[0019.13]
ORLD
ANDLD
ANDNOT 817.14  ; RK_07 #3托盘下料上升到位感应标志[0017.14]
OUT 617.14  ; RK_07 #3托盘下料电机正转[A]
LD TR0
LD D1113.00  ; RK_07 铝壳上料移载机构单步/自动循环运行中（总）
ANDNOT W242.12  ; RK_07 #3铝壳下料电机启动标志
ANDNOT H65.00  ; RK_07 铝壳托盘下料升降机构手动下料记忆
AND D1122.04  ; RK_07 铝壳上料移载机构#3铝壳托盘卸载电机反转3（步）
AND 865.03  ; RK_07 U8_Z 铝壳上料移载Y轴#3铝壳托盘下料位标志
AND H50.00  ; RK_07 U8_Z 铝壳上料移载Y轴回原点记忆
ANDNOT 117.02  ; RK_07 铝壳上料移载吸盘立真空
ANDNOT 817.02  ; RK_07 铝壳上料移载吸盘真空标志[0017.02]
ANDNOT H50.10  ; RK_07 铝壳上料移载机构吸盘立真空记忆
ANDNOT H51.00  ; RK_07 铝壳上料移载机构有料记忆
ANDNOT H51.10  ; RK_07 铝壳上料移载机构有托盘记忆
AND H66.00  ; RK_07 铝壳托盘下料升降机构有料记忆
ANDNOT 818.01  ; RK_07 #3托盘下料满托盘位（#2）标志[0018.01]
AND 817.14  ; RK_07 #3托盘下料上升到位感应标志[0017.14]
LD W1.01  ; 自动模式
OR W1.00  ; 手动模式
AND W242.12  ; RK_07 #3铝壳下料电机启动标志
AND H65.00  ; RK_07 铝壳托盘下料升降机构手动下料记忆
LD H66.00  ; RK_07 铝壳托盘下料升降机构有料记忆
AND H65.00  ; RK_07 铝壳托盘下料升降机构手动下料记忆
AND 814.12  ; RK_07 #3托盘下料车定位升降气缸上升位标志[0014.12]
AND 817.15  ; RK_07 #3托盘下料位物料车到位感应标志[0017.15]
AND 819.14  ; RK_07 #3托盘下料位物料车到位感应#2标志[0019.14]
ANDNOT 818.00  ; RK_07 #3托盘下料初始位（#1）标志[0018.00]
LD 819.13  ; RK_07 #3托盘下料下降到位感应标志[0019.13]
AND P_On
LDNOT P_On
AND 817.14  ; RK_07 #3托盘下料上升到位感应标志[0017.14]
ORLD
ANDNOT H66.00  ; RK_07 铝壳托盘下料升降机构有料记忆
AND H65.00  ; RK_07 铝壳托盘下料升降机构手动下料记忆
AND 814.13  ; RK_07 #3托盘下料车定位升降气缸下降位标志[0014.13]
ANDNOT 817.15  ; RK_07 #3托盘下料位物料车到位感应标志[0017.15]
ANDNOT 819.14  ; RK_07 #3托盘下料位物料车到位感应#2标志[0019.14]
AND T2615  ; #3铝壳下料电机初次下料反转到安全位延时
ORLD
ANDLD
ORLD
ANDLD
ANDNOT 117.14  ; RK_07 #3托盘下料电机正转
ANDNOT 117.15  ; RK_07 #3托盘下料电机反转
OUT 517.15  ; RK_07 #3托盘下料电机反转条件
TIMX(550) 0387 D18  ; 自动运行条件延时时间, RK_07 #3托盘下料电机反转延时[A]
LD TR0
LD D1113.00  ; RK_07 铝壳上料移载机构单步/自动循环运行中（总）
ANDNOT W242.12  ; RK_07 #3铝壳下料电机启动标志
ANDNOT H65.00  ; RK_07 铝壳托盘下料升降机构手动下料记忆
LD W1.01  ; 自动模式
OR W1.00  ; 手动模式
AND W242.12  ; RK_07 #3铝壳下料电机启动标志
AND H65.00  ; RK_07 铝壳托盘下料升降机构手动下料记忆
ORLD
ANDLD
LD 517.15  ; RK_07 #3托盘下料电机反转条件
AND T0387  ; RK_07 #3托盘下料电机反转延时[A]
OR 617.15  ; RK_07 #3托盘下料电机反传[A]
ANDLD
ANDNOT 818.00  ; RK_07 #3托盘下料初始位（#1）标志[0018.00]
LDNOT W242.12  ; RK_07 #3铝壳下料电机启动标志
ANDNOT H65.00  ; RK_07 铝壳托盘下料升降机构手动下料记忆
LD 819.13  ; RK_07 #3托盘下料下降到位感应标志[0019.13]
OR 817.14  ; RK_07 #3托盘下料上升到位感应标志[0017.14]
ANDLD
LD W242.12  ; RK_07 #3铝壳下料电机启动标志
AND H65.00  ; RK_07 铝壳托盘下料升降机构手动下料记忆
LD H66.00  ; RK_07 铝壳托盘下料升降机构有料记忆
ORNOT H66.00  ; RK_07 铝壳托盘下料升降机构有料记忆
ANDLD
ORLD
ANDLD
OUT 617.15  ; RK_07 #3托盘下料电机反传[A]

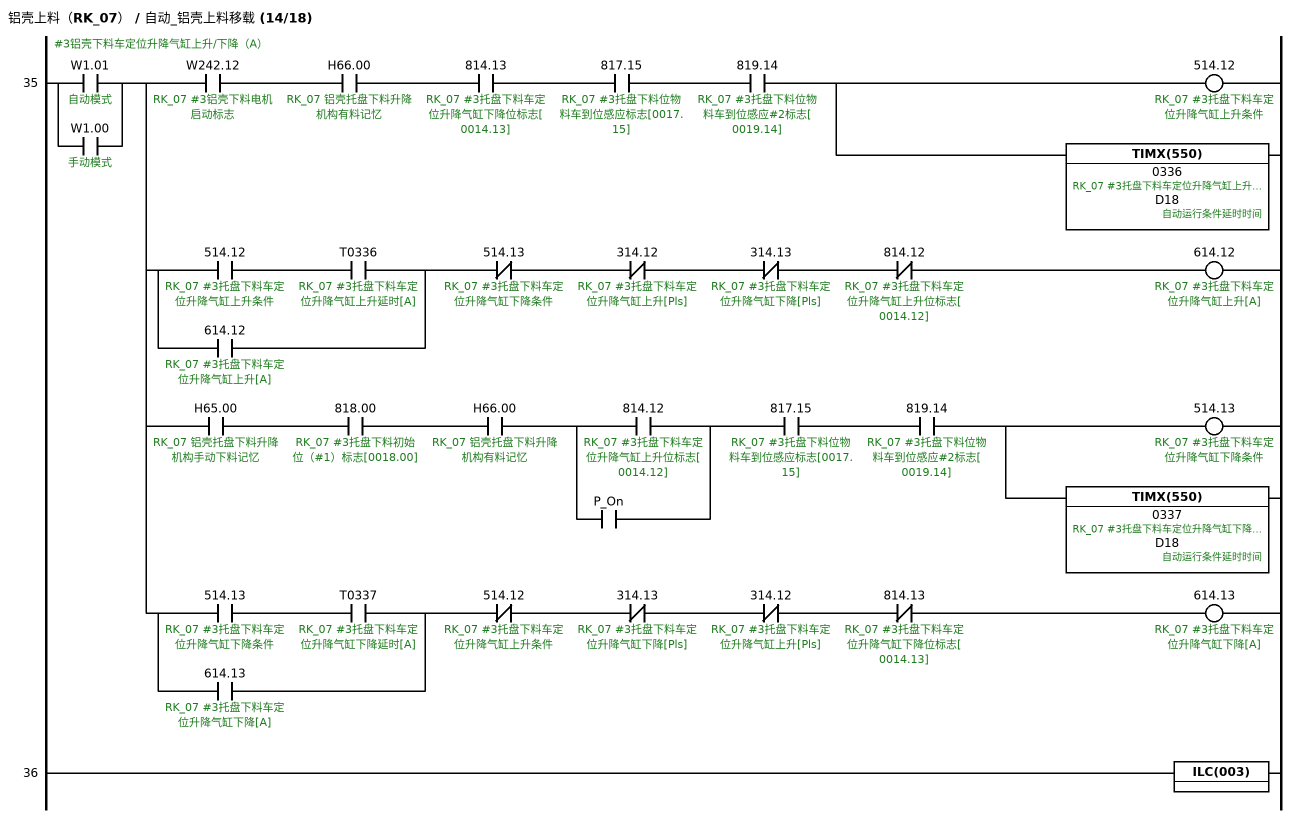
; rung 35: #3铝壳下料车定位升降气缸上升/下降（A）
LD W1.01  ; 自动模式
OR W1.00  ; 手动模式
OUT TR0
AND W242.12  ; RK_07 #3铝壳下料电机启动标志
AND H66.00  ; RK_07 铝壳托盘下料升降机构有料记忆
AND 814.13  ; RK_07 #3托盘下料车定位升降气缸下降位标志[0014.13]
AND 817.15  ; RK_07 #3托盘下料位物料车到位感应标志[0017.15]
AND 819.14  ; RK_07 #3托盘下料位物料车到位感应#2标志[0019.14]
OUT 514.12  ; RK_07 #3托盘下料车定位升降气缸上升条件
TIMX(550) 0336 D18  ; 自动运行条件延时时间, RK_07 #3托盘下料车定位升降气缸上升延时[A]
LD TR0
LD 514.12  ; RK_07 #3托盘下料车定位升降气缸上升条件
AND T0336  ; RK_07 #3托盘下料车定位升降气缸上升延时[A]
OR 614.12  ; RK_07 #3托盘下料车定位升降气缸上升[A]
ANDLD
ANDNOT 514.13  ; RK_07 #3托盘下料车定位升降气缸下降条件
ANDNOT 314.12  ; RK_07 #3托盘下料车定位升降气缸上升[Pls]
ANDNOT 314.13  ; RK_07 #3托盘下料车定位升降气缸下降[Pls]
ANDNOT 814.12  ; RK_07 #3托盘下料车定位升降气缸上升位标志[0014.12]
OUT 614.12  ; RK_07 #3托盘下料车定位升降气缸上升[A]
LD TR0
AND H65.00  ; RK_07 铝壳托盘下料升降机构手动下料记忆
AND 818.00  ; RK_07 #3托盘下料初始位（#1）标志[0018.00]
AND H66.00  ; RK_07 铝壳托盘下料升降机构有料记忆
LD 814.12  ; RK_07 #3托盘下料车定位升降气缸上升位标志[0014.12]
OR P_On
ANDLD
AND 817.15  ; RK_07 #3托盘下料位物料车到位感应标志[0017.15]
AND 819.14  ; RK_07 #3托盘下料位物料车到位感应#2标志[0019.14]
OUT 514.13  ; RK_07 #3托盘下料车定位升降气缸下降条件
TIMX(550) 0337 D18  ; 自动运行条件延时时间, RK_07 #3托盘下料车定位升降气缸下降延时[A]
LD TR0
LD 514.13  ; RK_07 #3托盘下料车定位升降气缸下降条件
AND T0337  ; RK_07 #3托盘下料车定位升降气缸下降延时[A]
OR 614.13  ; RK_07 #3托盘下料车定位升降气缸下降[A]
ANDLD
ANDNOT 514.12  ; RK_07 #3托盘下料车定位升降气缸上升条件
ANDNOT 314.13  ; RK_07 #3托盘下料车定位升降气缸下降[Pls]
ANDNOT 314.12  ; RK_07 #3托盘下料车定位升降气缸上升[Pls]
ANDNOT 814.13  ; RK_07 #3托盘下料车定位升降气缸下降位标志[0014.13]
OUT 614.13  ; RK_07 #3托盘下料车定位升降气缸下降[A]
; rung 36
ILC(003)

